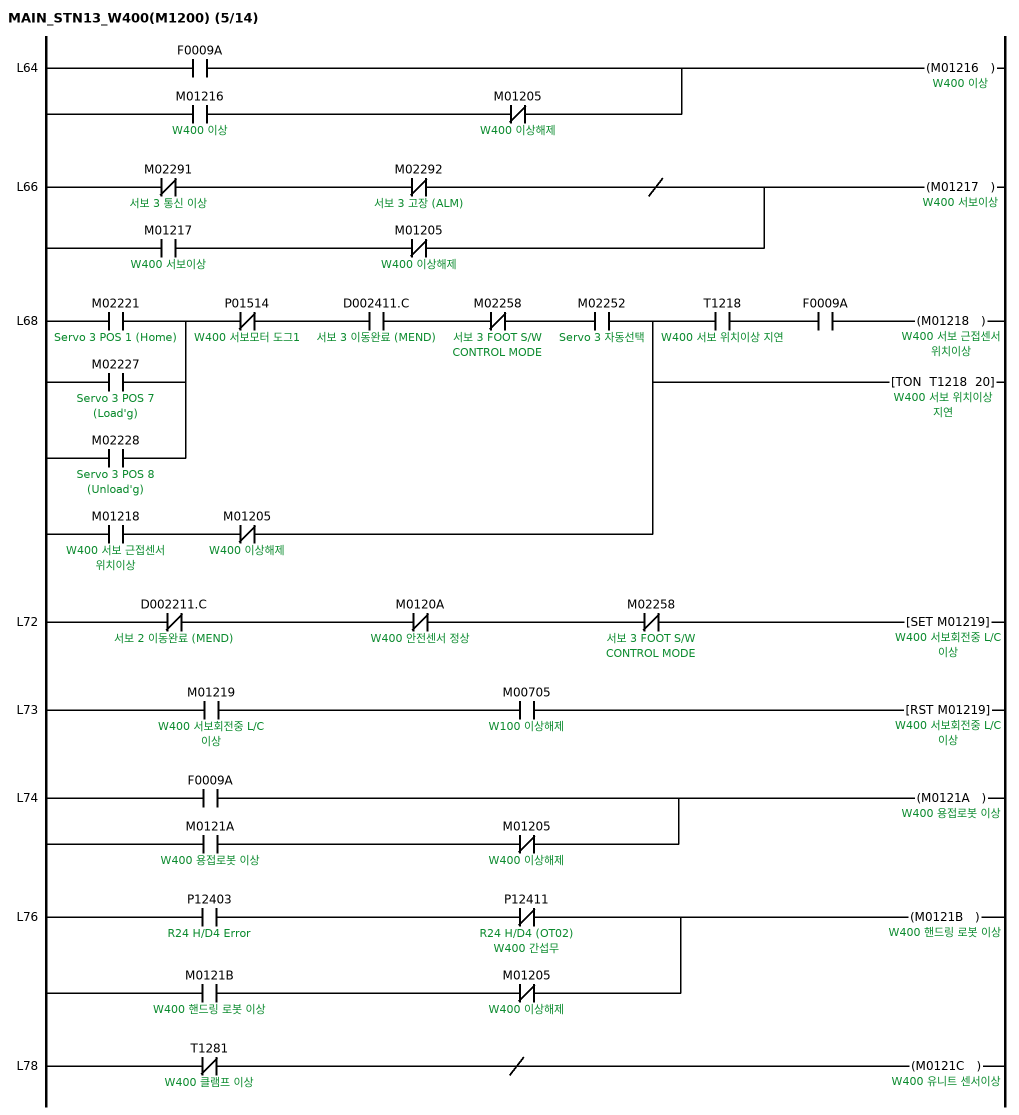
[picture p216: MAIN_STN13_W400(M1200) rungs L64-L78]
; L64
LOAD      F0009A
LOAD      M01216	// W400 이상
AND NOT   M01205	// W400 이상해제
OR LOAD
OUT       M01216	// W400 이상
; L66
LOAD NOT  M02291	// 서보 3 통신 이상
AND NOT   M02292	// 서보 3 고장 (ALM)
NOT
LOAD      M01217	// W400 서보이상
AND NOT   M01205	// W400 이상해제
OR LOAD
OUT       M01217	// W400 서보이상
; L68
LOAD      M02221	// Servo 3 POS 1 (Home)
OR        M02227	// Servo 3 POS 7 (Load'g)
OR        M02228	// Servo 3 POS 8 (Unload'g)
AND NOT   P01514	// W400 서보모터 도그1
AND       D002411.C	// 서보 3 이동완료 (MEND)
AND NOT   M02258	// 서보 3 FOOT S/W CONTROL MODE
AND       M02252	// Servo 3 자동선택
LOAD      M01218	// W400 서보 근접센서 위치이상
AND NOT   M01205	// W400 이상해제
OR LOAD
MPUSH
AND       T1218	// W400 서보 위치이상 지연
AND       F0009A
OUT       M01218	// W400 서보 근접센서 위치이상
MPOP
TON       T1218 20	// W400 서보 위치이상 지연
; L72
LOAD NOT  D002211.C	// 서보 2 이동완료 (MEND)
AND NOT   M0120A	// W400 안전센서 정상
AND NOT   M02258	// 서보 3 FOOT S/W CONTROL MODE
SET       M01219	// W400 서보회전중 L/C 이상
; L73
LOAD      M01219	// W400 서보회전중 L/C 이상
AND       M00705	// W100 이상해제
RST       M01219	// W400 서보회전중 L/C 이상
; L74
LOAD      F0009A
LOAD      M0121A	// W400 용접로봇 이상
AND NOT   M01205	// W400 이상해제
OR LOAD
OUT       M0121A	// W400 용접로봇 이상
; L76
LOAD      P12403	// R24 H/D4 Error
AND NOT   P12411	// R24 H/D4 (OT02) W400 간섭무
LOAD      M0121B	// W400 핸드링 로봇 이상
AND NOT   M01205	// W400 이상해제
OR LOAD
OUT       M0121B	// W400 핸드링 로봇 이상
; L78
LOAD NOT  T1281	// W400 클램프 이상
NOT
OUT       M0121C	// W400 유니트 센서이상

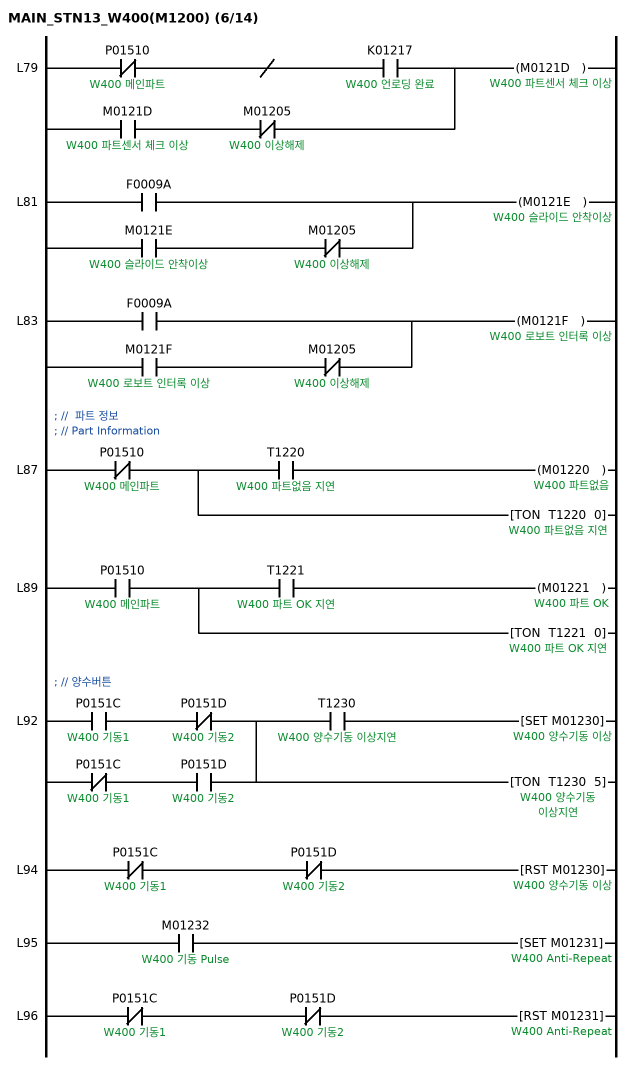
; L79
LOAD NOT  P01510	// W400 메인파트
NOT
AND       K01217	// W400 언로딩 완료
LOAD      M0121D	// W400 파트센서 체크 이상
AND NOT   M01205	// W400 이상해제
OR LOAD
OUT       M0121D	// W400 파트센서 체크 이상
; L81
LOAD      F0009A
LOAD      M0121E	// W400 슬라이드 안착이상
AND NOT   M01205	// W400 이상해제
OR LOAD
OUT       M0121E	// W400 슬라이드 안착이상
; L83
LOAD      F0009A
LOAD      M0121F	// W400 로보트 인터록 이상
AND NOT   M01205	// W400 이상해제
OR LOAD
OUT       M0121F	// W400 로보트 인터록 이상
//   //  파트 정보
//   // Part Information
; L87
LOAD NOT  P01510	// W400 메인파트
MPUSH
AND       T1220	// W400 파트없음 지연
OUT       M01220	// W400 파트없음
MPOP
TON       T1220 0	// W400 파트없음 지연
; L89
LOAD      P01510	// W400 메인파트
MPUSH
AND       T1221	// W400 파트 OK 지연
OUT       M01221	// W400 파트 OK
MPOP
TON       T1221 0	// W400 파트 OK 지연
//   // 양수버튼
; L92
LOAD      P0151C	// W400 기동1
AND NOT   P0151D	// W400 기동2
LOAD NOT  P0151C	// W400 기동1
AND       P0151D	// W400 기동2
OR LOAD
MPUSH
AND       T1230	// W400 양수기동 이상지연
SET       M01230	// W400 양수기동 이상
MPOP
TON       T1230 5	// W400 양수기동 이상지연
; L94
LOAD NOT  P0151C	// W400 기동1
AND NOT   P0151D	// W400 기동2
RST       M01230	// W400 양수기동 이상
; L95
LOAD      M01232	// W400 기동 Pulse
SET       M01231	// W400 Anti-Repeat
; L96
LOAD NOT  P0151C	// W400 기동1
AND NOT   P0151D	// W400 기동2
RST       M01231	// W400 Anti-Repeat

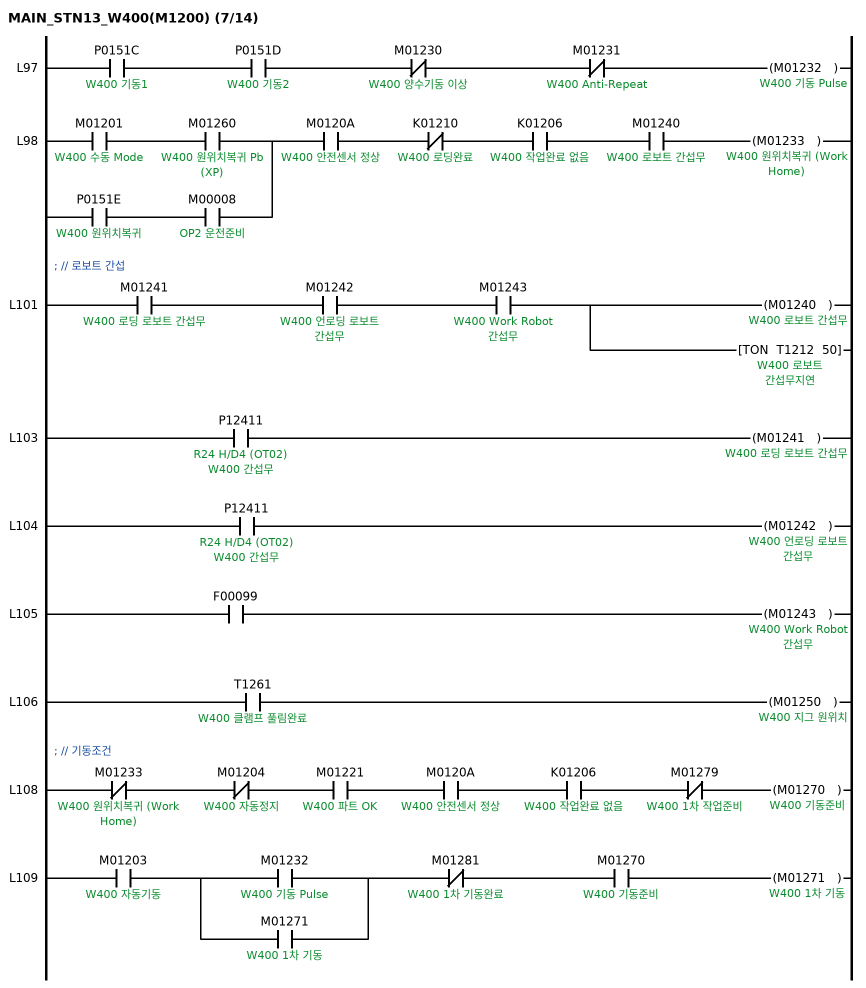
; L97
LOAD      P0151C	// W400 기동1
AND       P0151D	// W400 기동2
AND NOT   M01230	// W400 양수기동 이상
AND NOT   M01231	// W400 Anti-Repeat
OUT       M01232	// W400 기동 Pulse
; L98
LOAD      M01201	// W400 수동 Mode
AND       M01260	// W400 원위치복귀 Pb (XP)
LOAD      P0151E	// W400 원위치복귀
AND       M00008	// OP2 운전준비
OR LOAD
AND       M0120A	// W400 안전센서 정상
AND NOT   K01210	// W400 로딩완료
AND       K01206	// W400 작업완료 없음
AND       M01240	// W400 로보트 간섭무
OUT       M01233	// W400 원위치복귀 (Work Home)
//   // 로보트 간섭
; L101
LOAD      M01241	// W400 로딩 로보트 간섭무
AND       M01242	// W400 언로딩 로보트 간섭무
AND       M01243	// W400 Work Robot 간섭무
OUT       M01240	// W400 로보트 간섭무
TON       T1212 50	// W400 로보트 간섭무지연
; L103
LOAD      P12411	// R24 H/D4 (OT02) W400 간섭무
OUT       M01241	// W400 로딩 로보트 간섭무
; L104
LOAD      P12411	// R24 H/D4 (OT02) W400 간섭무
OUT       M01242	// W400 언로딩 로보트 간섭무
; L105
LOAD      F00099
OUT       M01243	// W400 Work Robot 간섭무
; L106
LOAD      T1261	// W400 클램프 풀림완료
OUT       M01250	// W400 지그 원위치
//   // 기동조건
; L108
LOAD NOT  M01233	// W400 원위치복귀 (Work Home)
AND NOT   M01204	// W400 자동정지
AND       M01221	// W400 파트 OK
AND       M0120A	// W400 안전센서 정상
AND       K01206	// W400 작업완료 없음
AND NOT   M01279	// W400 1차 작업준비
OUT       M01270	// W400 기동준비
; L109
LOAD      M01203	// W400 자동기동
LOAD      M01232	// W400 기동 Pulse
OR        M01271	// W400 1차 기동
AND LOAD
AND NOT   M01281	// W400 1차 기동완료
AND       M01270	// W400 기동준비
OUT       M01271	// W400 1차 기동

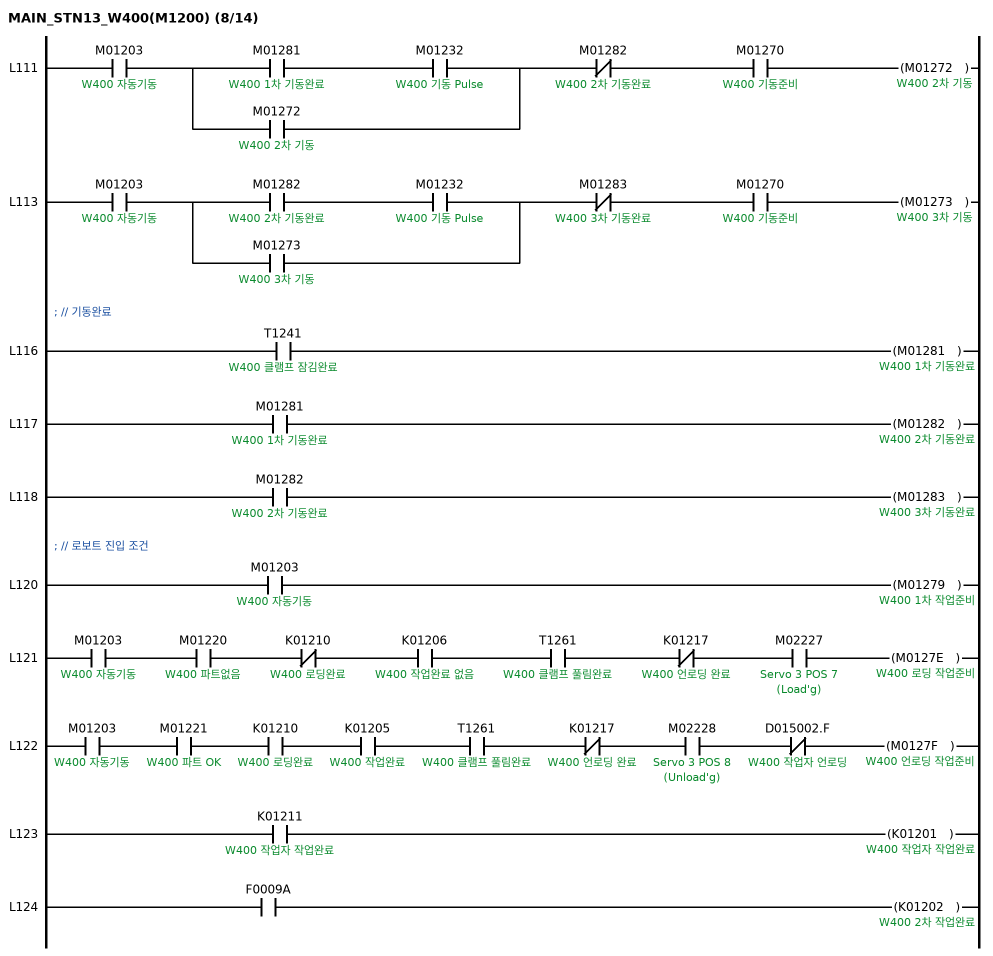
; L111
LOAD      M01203	// W400 자동기동
LOAD      M01281	// W400 1차 기동완료
AND       M01232	// W400 기동 Pulse
OR        M01272	// W400 2차 기동
AND LOAD
AND NOT   M01282	// W400 2차 기동완료
AND       M01270	// W400 기동준비
OUT       M01272	// W400 2차 기동
; L113
LOAD      M01203	// W400 자동기동
LOAD      M01282	// W400 2차 기동완료
AND       M01232	// W400 기동 Pulse
OR        M01273	// W400 3차 기동
AND LOAD
AND NOT   M01283	// W400 3차 기동완료
AND       M01270	// W400 기동준비
OUT       M01273	// W400 3차 기동
//   // 기동완료
; L116
LOAD      T1241	// W400 클램프 잠김완료
OUT       M01281	// W400 1차 기동완료
; L117
LOAD      M01281	// W400 1차 기동완료
OUT       M01282	// W400 2차 기동완료
; L118
LOAD      M01282	// W400 2차 기동완료
OUT       M01283	// W400 3차 기동완료
//   // 로보트 진입 조건
; L120
LOAD      M01203	// W400 자동기동
OUT       M01279	// W400 1차 작업준비
; L121
LOAD      M01203	// W400 자동기동
AND       M01220	// W400 파트없음
AND NOT   K01210	// W400 로딩완료
AND       K01206	// W400 작업완료 없음
AND       T1261	// W400 클램프 풀림완료
AND NOT   K01217	// W400 언로딩 완료
AND       M02227	// Servo 3 POS 7 (Load'g)
OUT       M0127E	// W400 로딩 작업준비
; L122
LOAD      M01203	// W400 자동기동
AND       M01221	// W400 파트 OK
AND       K01210	// W400 로딩완료
AND       K01205	// W400 작업완료
AND       T1261	// W400 클램프 풀림완료
AND NOT   K01217	// W400 언로딩 완료
AND       M02228	// Servo 3 POS 8 (Unload'g)
AND NOT   D015002.F	// W400 작업자 언로딩
OUT       M0127F	// W400 언로딩 작업준비
; L123
LOAD      K01211	// W400 작업자 작업완료
OUT       K01201	// W400 작업자 작업완료
; L124
LOAD      F0009A
OUT       K01202	// W400 2차 작업완료

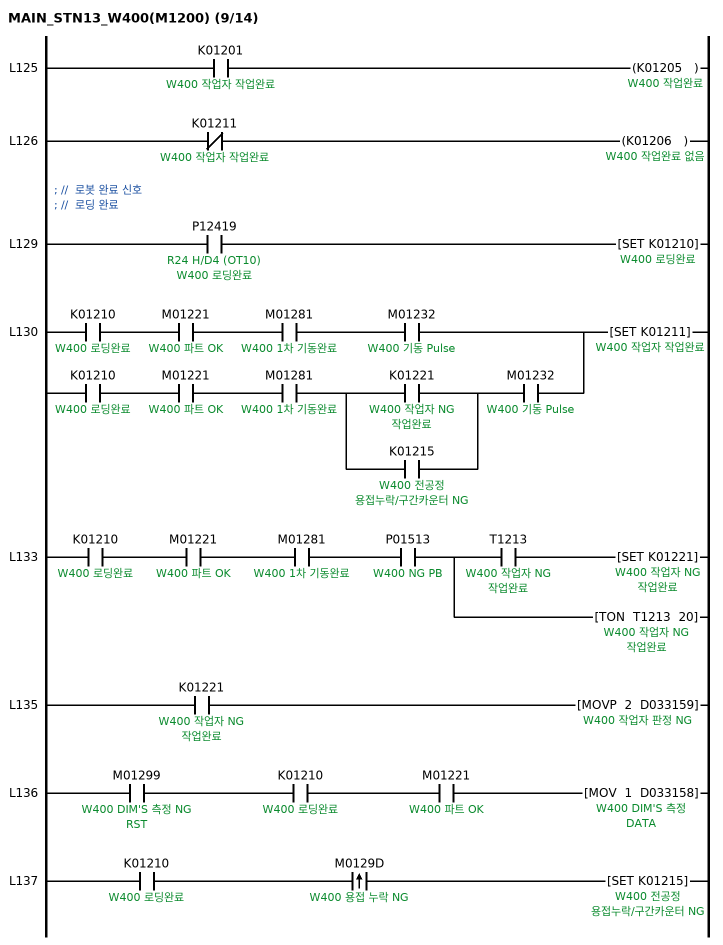
; L125
LOAD      K01201	// W400 작업자 작업완료
OUT       K01205	// W400 작업완료
; L126
LOAD NOT  K01211	// W400 작업자 작업완료
OUT       K01206	// W400 작업완료 없음
//   //  로봇 완료 신호
//   //  로딩 완료
; L129
LOAD      P12419	// R24 H/D4 (OT10) W400 로딩완료
SET       K01210	// W400 로딩완료
; L130
LOAD      K01210	// W400 로딩완료
AND       M01221	// W400 파트 OK
AND       M01281	// W400 1차 기동완료
AND       M01232	// W400 기동 Pulse
LOAD      K01210	// W400 로딩완료
AND       M01221	// W400 파트 OK
AND       M01281	// W400 1차 기동완료
LOAD      K01221	// W400 작업자 NG 작업완료
OR        K01215	// W400 전공정 용접누락/구간카운터 NG
AND LOAD
AND       M01232	// W400 기동 Pulse
OR LOAD
SET       K01211	// W400 작업자 작업완료
; L133
LOAD      K01210	// W400 로딩완료
AND       M01221	// W400 파트 OK
AND       M01281	// W400 1차 기동완료
AND       P01513	// W400 NG PB
MPUSH
AND       T1213	// W400 작업자 NG 작업완료
SET       K01221	// W400 작업자 NG 작업완료
MPOP
TON       T1213 20	// W400 작업자 NG 작업완료
; L135
LOAD      K01221	// W400 작업자 NG 작업완료
MOVP      2 D033159	// W400 작업자 판정 NG
; L136
LOAD      M01299	// W400 DIM'S 측정 NG RST
AND       K01210	// W400 로딩완료
AND       M01221	// W400 파트 OK
MOV       1 D033158	// W400 DIM'S 측정 DATA
; L137
LOAD      K01210	// W400 로딩완료
ANDP      M0129D	// W400 용접 누락 NG
SET       K01215	// W400 전공정 용접누락/구간카운터 NG

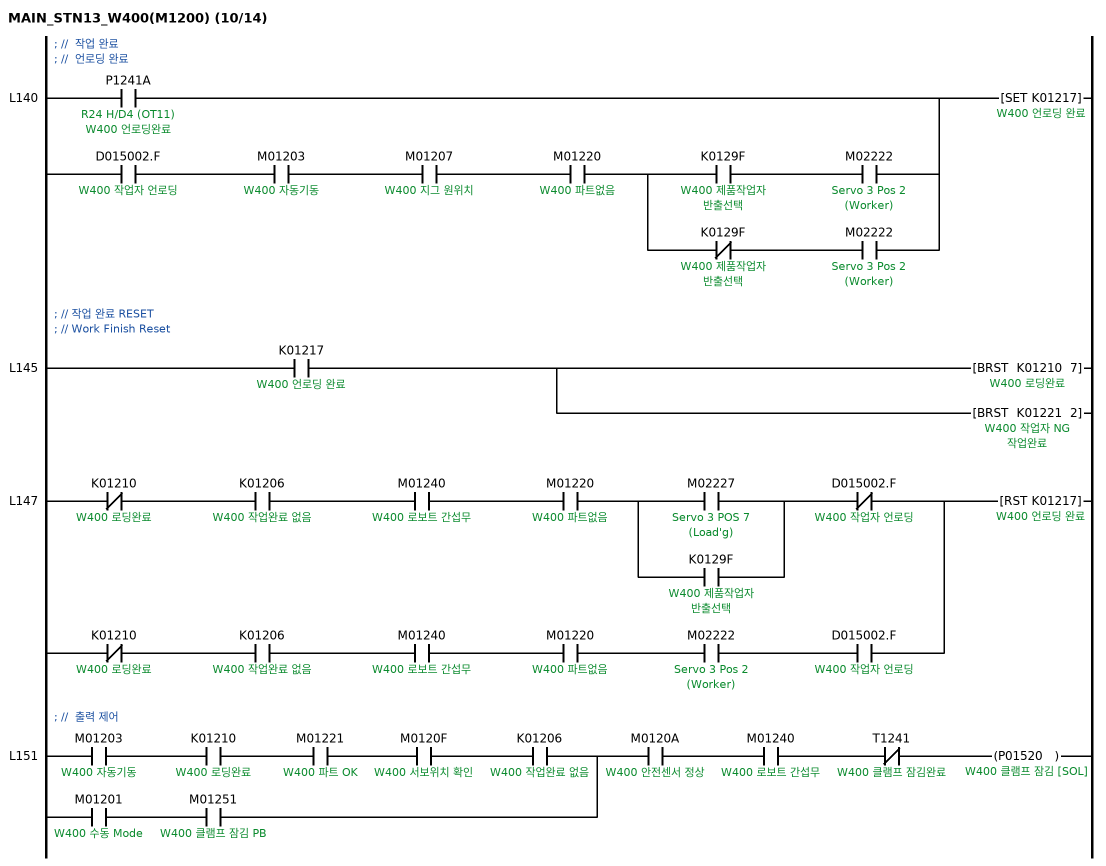
//   //  작업 완료
//   //  언로딩 완료
; L140
LOAD      P1241A	// R24 H/D4 (OT11) W400 언로딩완료
LOAD      D015002.F	// W400 작업자 언로딩
AND       M01203	// W400 자동기동
AND       M01207	// W400 지그 원위치
AND       M01220	// W400 파트없음
LOAD      K0129F	// W400 제품작업자 반출선택
AND       M02222	// Servo 3 Pos 2 (Worker)
LOAD NOT  K0129F	// W400 제품작업자 반출선택
AND       M02222	// Servo 3 Pos 2 (Worker)
OR LOAD
AND LOAD
OR LOAD
SET       K01217	// W400 언로딩 완료
//     // 작업 완료 RESET
//   // Work Finish Reset
; L145
LOAD      K01217	// W400 언로딩 완료
BRST      K01210 7	// W400 로딩완료
BRST      K01221 2	// W400 작업자 NG 작업완료
; L147
LOAD NOT  K01210	// W400 로딩완료
AND       K01206	// W400 작업완료 없음
AND       M01240	// W400 로보트 간섭무
AND       M01220	// W400 파트없음
LOAD      M02227	// Servo 3 POS 7 (Load'g)
OR        K0129F	// W400 제품작업자 반출선택
AND LOAD
AND NOT   D015002.F	// W400 작업자 언로딩
LOAD NOT  K01210	// W400 로딩완료
AND       K01206	// W400 작업완료 없음
AND       M01240	// W400 로보트 간섭무
AND       M01220	// W400 파트없음
AND       M02222	// Servo 3 Pos 2 (Worker)
AND       D015002.F	// W400 작업자 언로딩
OR LOAD
RST       K01217	// W400 언로딩 완료
//     //  출력 제어
; L151
LOAD      M01203	// W400 자동기동
AND       K01210	// W400 로딩완료
AND       M01221	// W400 파트 OK
AND       M0120F	// W400 서보위치 확인
AND       K01206	// W400 작업완료 없음
LOAD      M01201	// W400 수동 Mode
AND       M01251	// W400 클램프 잠김 PB
OR LOAD
AND       M0120A	// W400 안전센서 정상
AND       M01240	// W400 로보트 간섭무
AND NOT   T1241	// W400 클램프 잠김완료
OUT       P01520	// W400 클램프 잠김 [SOL]

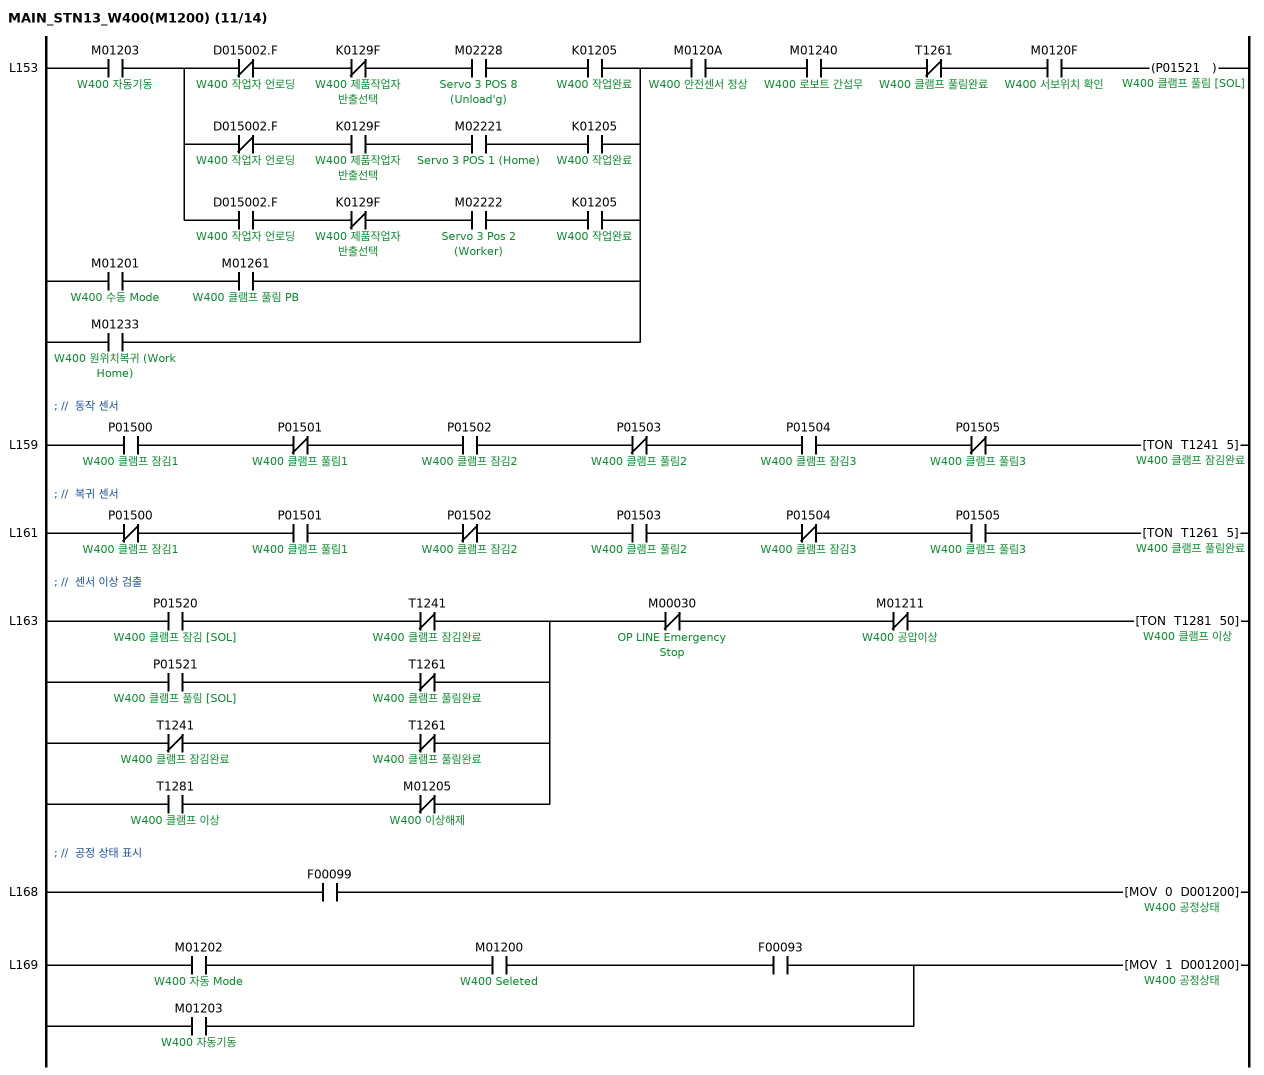
; L153
LOAD      M01203	// W400 자동기동
LOAD NOT  D015002.F	// W400 작업자 언로딩
AND NOT   K0129F	// W400 제품작업자 반출선택
AND       M02228	// Servo 3 POS 8 (Unload'g)
AND       K01205	// W400 작업완료
LOAD NOT  D015002.F	// W400 작업자 언로딩
AND       K0129F	// W400 제품작업자 반출선택
AND       M02221	// Servo 3 POS 1 (Home)
AND       K01205	// W400 작업완료
OR LOAD
LOAD      D015002.F	// W400 작업자 언로딩
AND NOT   K0129F	// W400 제품작업자 반출선택
AND       M02222	// Servo 3 Pos 2 (Worker)
AND       K01205	// W400 작업완료
OR LOAD
AND LOAD
LOAD      M01201	// W400 수동 Mode
AND       M01261	// W400 클램프 풀림 PB
OR LOAD
OR        M01233	// W400 원위치복귀 (Work Home)
AND       M0120A	// W400 안전센서 정상
AND       M01240	// W400 로보트 간섭무
AND NOT   T1261	// W400 클램프 풀림완료
AND       M0120F	// W400 서보위치 확인
OUT       P01521	// W400 클램프 풀림 [SOL]
//   //  동작 센서
; L159
LOAD      P01500	// W400 클램프 잠김1
AND NOT   P01501	// W400 클램프 풀림1
AND       P01502	// W400 클램프 잠김2
AND NOT   P01503	// W400 클램프 풀림2
AND       P01504	// W400 클램프 잠김3
AND NOT   P01505	// W400 클램프 풀림3
TON       T1241 5	// W400 클램프 잠김완료
//   //  복귀 센서
; L161
LOAD NOT  P01500	// W400 클램프 잠김1
AND       P01501	// W400 클램프 풀림1
AND NOT   P01502	// W400 클램프 잠김2
AND       P01503	// W400 클램프 풀림2
AND NOT   P01504	// W400 클램프 잠김3
AND       P01505	// W400 클램프 풀림3
TON       T1261 5	// W400 클램프 풀림완료
//     //  센서 이상 검출
; L163
LOAD      P01520	// W400 클램프 잠김 [SOL]
AND NOT   T1241	// W400 클램프 잠김완료
LOAD      P01521	// W400 클램프 풀림 [SOL]
AND NOT   T1261	// W400 클램프 풀림완료
OR LOAD
LOAD NOT  T1241	// W400 클램프 잠김완료
AND NOT   T1261	// W400 클램프 풀림완료
OR LOAD
LOAD      T1281	// W400 클램프 이상
AND NOT   M01205	// W400 이상해제
OR LOAD
AND NOT   M00030	// OP LINE Emergency Stop
AND NOT   M01211	// W400 공압이상
TON       T1281 50	// W400 클램프 이상
//   //  공정 상태 표시
; L168
LOAD      F00099
MOV       0 D001200	// W400 공정상태
; L169
LOAD      M01202	// W400 자동 Mode
AND       M01200	// W400 Seleted
AND       F00093
OR        M01203	// W400 자동기동
MOV       1 D001200	// W400 공정상태

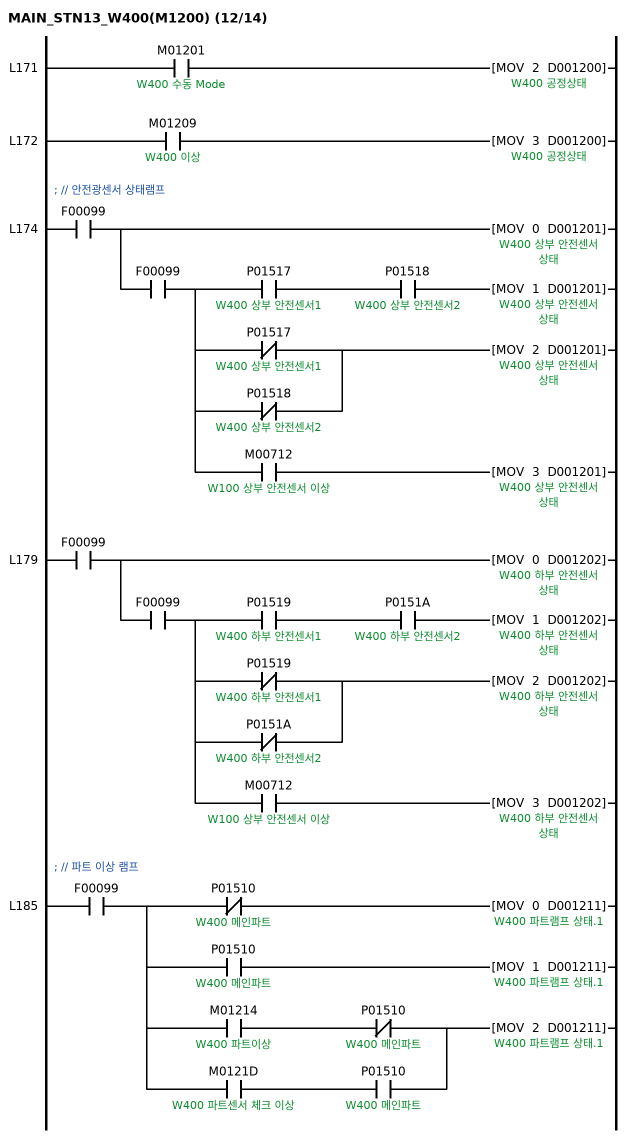
; L171
LOAD      M01201	// W400 수동 Mode
MOV       2 D001200	// W400 공정상태
; L172
LOAD      M01209	// W400 이상
MOV       3 D001200	// W400 공정상태
//   // 안전광센서 상태램프
; L174
LOAD      F00099
MOV       0 D001201	// W400 상부 안전센서 상태
AND       F00099
MPUSH
AND       P01517	// W400 상부 안전센서1
AND       P01518	// W400 상부 안전센서2
MOV       1 D001201	// W400 상부 안전센서 상태
MLOAD
LOAD NOT  P01517	// W400 상부 안전센서1
OR NOT    P01518	// W400 상부 안전센서2
AND LOAD
MOV       2 D001201	// W400 상부 안전센서 상태
MPOP
AND       M00712	// W100 상부 안전센서 이상
MOV       3 D001201	// W400 상부 안전센서 상태
; L179
LOAD      F00099
MOV       0 D001202	// W400 하부 안전센서 상태
AND       F00099
MPUSH
AND       P01519	// W400 하부 안전센서1
AND       P0151A	// W400 하부 안전센서2
MOV       1 D001202	// W400 하부 안전센서 상태
MLOAD
LOAD NOT  P01519	// W400 하부 안전센서1
OR NOT    P0151A	// W400 하부 안전센서2
AND LOAD
MOV       2 D001202	// W400 하부 안전센서 상태
MPOP
AND       M00712	// W100 상부 안전센서 이상
MOV       3 D001202	// W400 하부 안전센서 상태
//   // 파트 이상 램프
; L185
LOAD      F00099
MPUSH
AND NOT   P01510	// W400 메인파트
MOV       0 D001211	// W400 파트램프 상태.1
MLOAD
AND       P01510	// W400 메인파트
MOV       1 D001211	// W400 파트램프 상태.1
MPOP
LOAD      M01214	// W400 파트이상
AND NOT   P01510	// W400 메인파트
LOAD      M0121D	// W400 파트센서 체크 이상
AND       P01510	// W400 메인파트
OR LOAD
AND LOAD
MOV       2 D001211	// W400 파트램프 상태.1

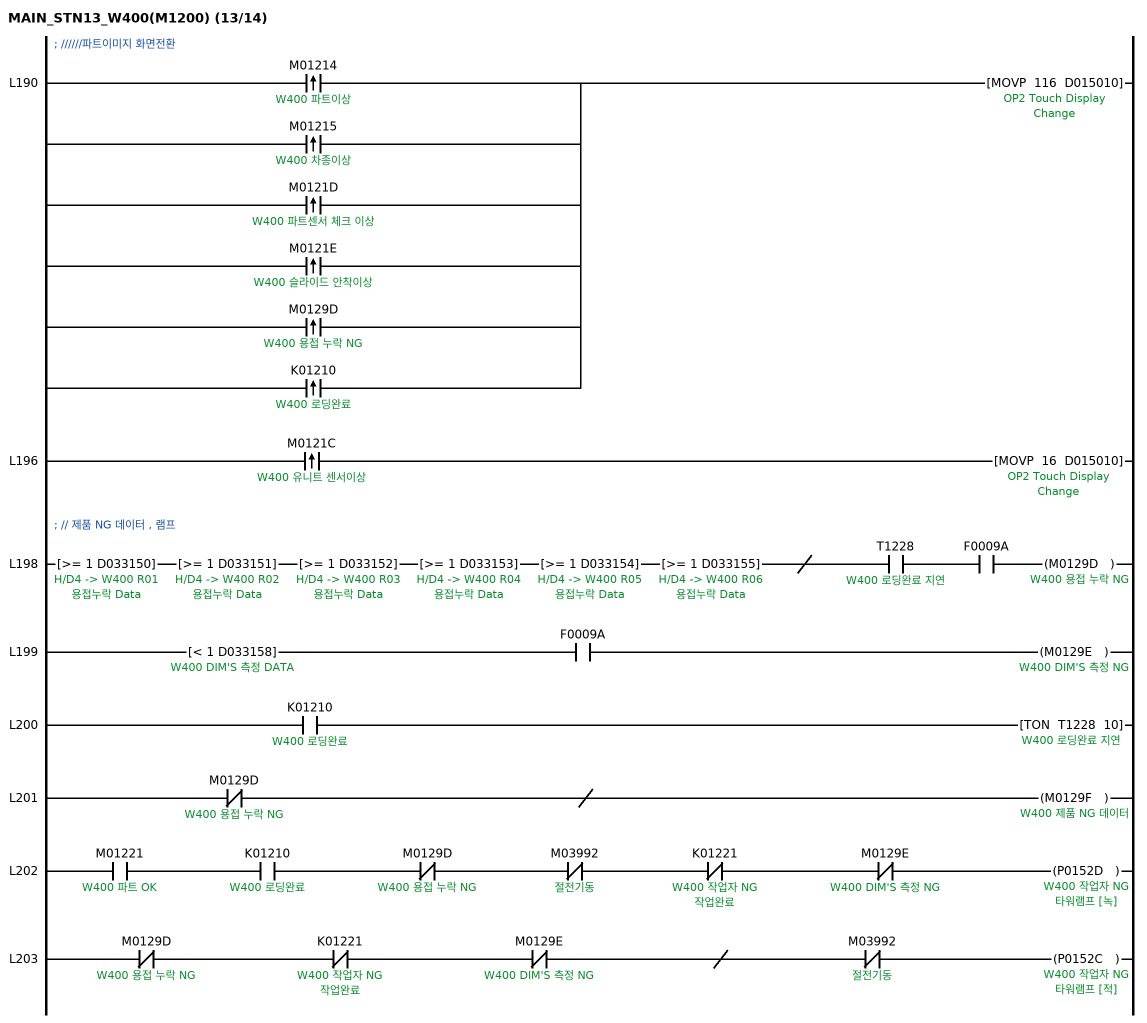
// //////파트이미지 화면전환
; L190
LOADP     M01214	// W400 파트이상
ORP       M01215	// W400 차종이상
ORP       M0121D	// W400 파트센서 체크 이상
ORP       M0121E	// W400 슬라이드 안착이상
ORP       M0129D	// W400 용접 누락 NG
ORP       K01210	// W400 로딩완료
MOVP      116 D015010	// OP2 Touch Display Change
; L196
LOADP     M0121C	// W400 유니트 센서이상
MOVP      16 D015010	// OP2 Touch Display Change
//   // 제품 NG 데이터 , 램프
; L198
LOAD>=    1 D033150	// H/D4 -> W400 R01 용접누락 Data
AND>=     1 D033151	// H/D4 -> W400 R02 용접누락 Data
AND>=     1 D033152	// H/D4 -> W400 R03 용접누락 Data
AND>=     1 D033153	// H/D4 -> W400 R04 용접누락 Data
AND>=     1 D033154	// H/D4 -> W400 R05 용접누락 Data
AND>=     1 D033155	// H/D4 -> W400 R06 용접누락 Data
NOT
AND       T1228	// W400 로딩완료 지연
AND       F0009A
OUT       M0129D	// W400 용접 누락 NG
; L199
LOAD<     1 D033158	// W400 DIM'S 측정 DATA
AND       F0009A
OUT       M0129E	// W400 DIM'S 측정 NG
; L200
LOAD      K01210	// W400 로딩완료
TON       T1228 10	// W400 로딩완료 지연
; L201
LOAD NOT  M0129D	// W400 용접 누락 NG
NOT
OUT       M0129F	// W400 제품 NG 데이터
; L202
LOAD      M01221	// W400 파트 OK
AND       K01210	// W400 로딩완료
AND NOT   M0129D	// W400 용접 누락 NG
AND NOT   M03992	// 절전기동
AND NOT   K01221	// W400 작업자 NG 작업완료
AND NOT   M0129E	// W400 DIM'S 측정 NG
OUT       P0152D	// W400 작업자 NG 타워램프 [녹]
; L203
LOAD NOT  M0129D	// W400 용접 누락 NG
AND NOT   K01221	// W400 작업자 NG 작업완료
AND NOT   M0129E	// W400 DIM'S 측정 NG
NOT
AND NOT   M03992	// 절전기동
OUT       P0152C	// W400 작업자 NG 타워램프 [적]

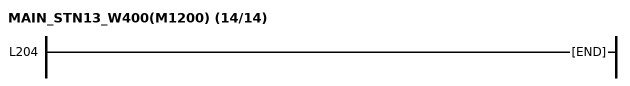
; L204
END

PROGRAM MAIN_STN14_W450(M1300) (task: 스캔 프로그램)

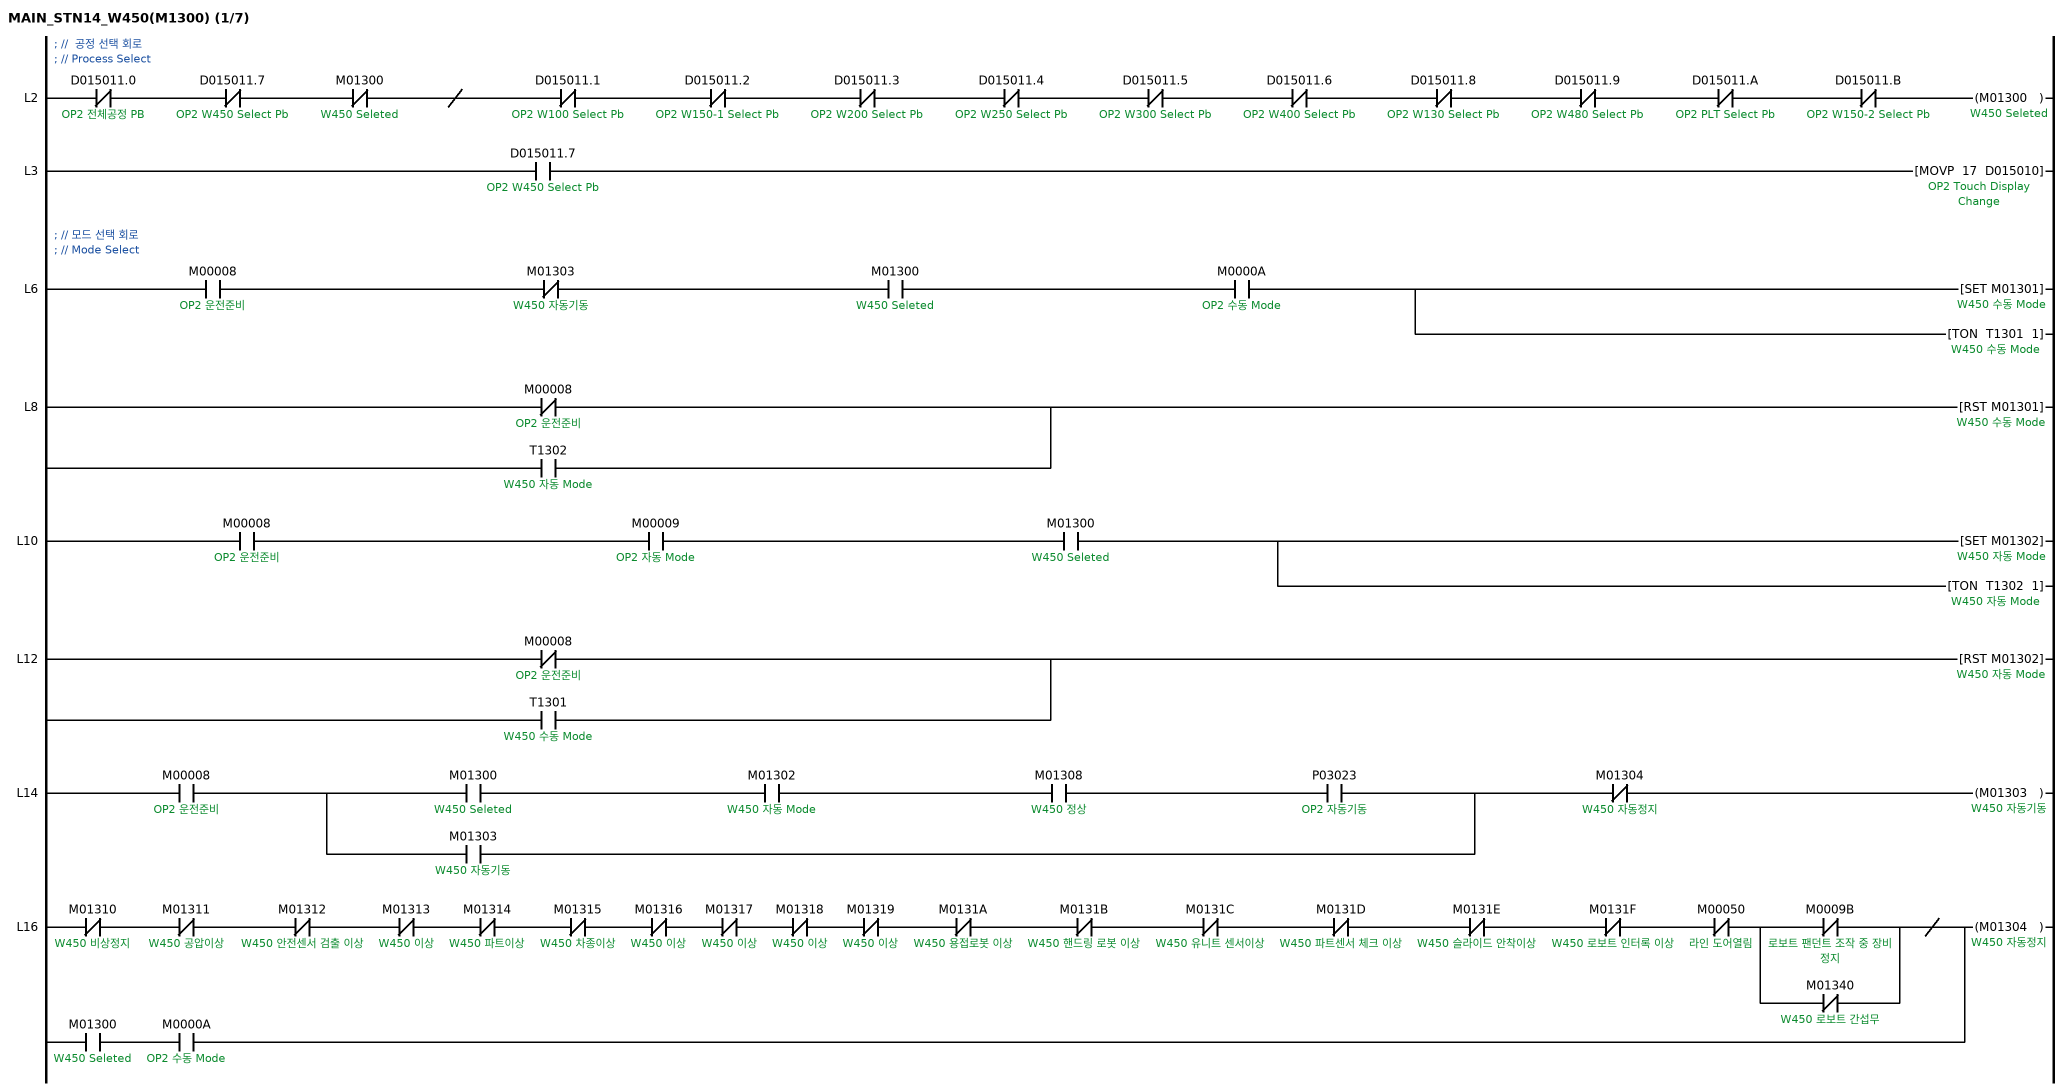
//   //  공정 선택 회로
//   // Process Select
; L2
LOAD NOT  D015011.0	// OP2 전체공정 PB
AND NOT   D015011.7	// OP2 W450 Select Pb
AND NOT   M01300	// W450 Seleted
NOT
AND NOT   D015011.1	// OP2 W100 Select Pb
AND NOT   D015011.2	// OP2 W150-1 Select Pb
AND NOT   D015011.3	// OP2 W200 Select Pb
AND NOT   D015011.4	// OP2 W250 Select Pb
AND NOT   D015011.5	// OP2 W300 Select Pb
AND NOT   D015011.6	// OP2 W400 Select Pb
AND NOT   D015011.8	// OP2 W130 Select Pb
AND NOT   D015011.9	// OP2 W480 Select Pb
AND NOT   D015011.A	// OP2 PLT Select Pb
AND NOT   D015011.B	// OP2 W150-2 Select Pb
OUT       M01300	// W450 Seleted
; L3
LOAD      D015011.7	// OP2 W450 Select Pb
MOVP      17 D015010	// OP2 Touch Display Change
// // 모드 선택 회로
//   // Mode Select
; L6
LOAD      M00008	// OP2 운전준비
AND NOT   M01303	// W450 자동기동
AND       M01300	// W450 Seleted
AND       M0000A	// OP2 수동 Mode
SET       M01301	// W450 수동 Mode
TON       T1301 1	// W450 수동 Mode
; L8
LOAD NOT  M00008	// OP2 운전준비
OR        T1302	// W450 자동 Mode
RST       M01301	// W450 수동 Mode
; L10
LOAD      M00008	// OP2 운전준비
AND       M00009	// OP2 자동 Mode
AND       M01300	// W450 Seleted
SET       M01302	// W450 자동 Mode
TON       T1302 1	// W450 자동 Mode
; L12
LOAD NOT  M00008	// OP2 운전준비
OR        T1301	// W450 수동 Mode
RST       M01302	// W450 자동 Mode
; L14
LOAD      M00008	// OP2 운전준비
LOAD      M01300	// W450 Seleted
AND       M01302	// W450 자동 Mode
AND       M01308	// W450 정상
AND       P03023	// OP2 자동기동
OR        M01303	// W450 자동기동
AND LOAD
AND NOT   M01304	// W450 자동정지
OUT       M01303	// W450 자동기동
; L16
LOAD NOT  M01310	// W450 비상정지
AND NOT   M01311	// W450 공압이상
AND NOT   M01312	// W450 안전센서 검출 이상
AND NOT   M01313	// W450 이상
AND NOT   M01314	// W450 파트이상
AND NOT   M01315	// W450 차종이상
AND NOT   M01316	// W450 이상
AND NOT   M01317	// W450 이상
AND NOT   M01318	// W450 이상
AND NOT   M01319	// W450 이상
AND NOT   M0131A	// W450 용접로봇 이상
AND NOT   M0131B	// W450 핸드링 로봇 이상
AND NOT   M0131C	// W450 유니트 센서이상
AND NOT   M0131D	// W450 파트센서 체크 이상
AND NOT   M0131E	// W450 슬라이드 안착이상
AND NOT   M0131F	// W450 로보트 인터록 이상
AND NOT   M00050	// 라인 도어열림
LOAD NOT  M0009B	// 로보트 팬던트 조작 중 장비 정지
OR NOT    M01340	// W450 로보트 간섭무
AND LOAD
NOT
LOAD      M01300	// W450 Seleted
AND       M0000A	// OP2 수동 Mode
OR LOAD
OUT       M01304	// W450 자동정지

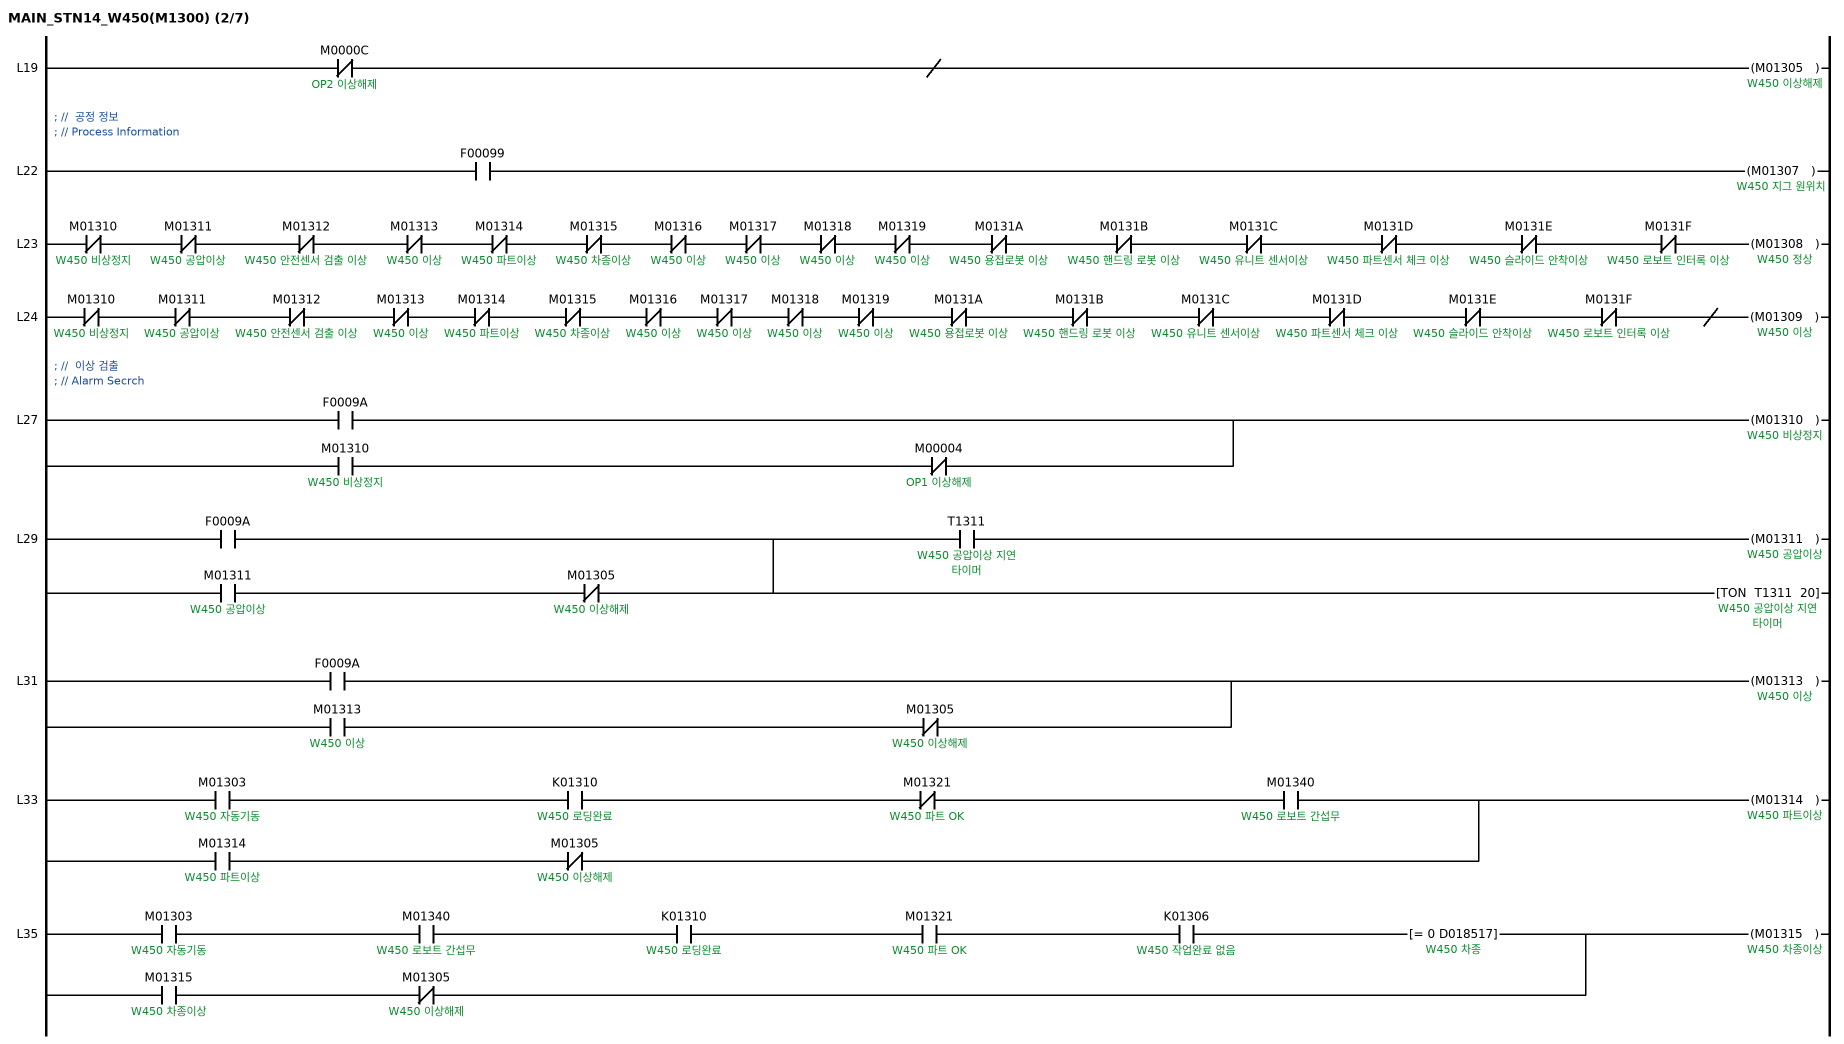
; L19
LOAD NOT  M0000C	// OP2 이상해제
NOT
OUT       M01305	// W450 이상해제
//   //  공정 정보
//   // Process Information
; L22
LOAD      F00099
OUT       M01307	// W450 지그 원위치
; L23
LOAD NOT  M01310	// W450 비상정지
AND NOT   M01311	// W450 공압이상
AND NOT   M01312	// W450 안전센서 검출 이상
AND NOT   M01313	// W450 이상
AND NOT   M01314	// W450 파트이상
AND NOT   M01315	// W450 차종이상
AND NOT   M01316	// W450 이상
AND NOT   M01317	// W450 이상
AND NOT   M01318	// W450 이상
AND NOT   M01319	// W450 이상
AND NOT   M0131A	// W450 용접로봇 이상
AND NOT   M0131B	// W450 핸드링 로봇 이상
AND NOT   M0131C	// W450 유니트 센서이상
AND NOT   M0131D	// W450 파트센서 체크 이상
AND NOT   M0131E	// W450 슬라이드 안착이상
AND NOT   M0131F	// W450 로보트 인터록 이상
OUT       M01308	// W450 정상
; L24
LOAD NOT  M01310	// W450 비상정지
AND NOT   M01311	// W450 공압이상
AND NOT   M01312	// W450 안전센서 검출 이상
AND NOT   M01313	// W450 이상
AND NOT   M01314	// W450 파트이상
AND NOT   M01315	// W450 차종이상
AND NOT   M01316	// W450 이상
AND NOT   M01317	// W450 이상
AND NOT   M01318	// W450 이상
AND NOT   M01319	// W450 이상
AND NOT   M0131A	// W450 용접로봇 이상
AND NOT   M0131B	// W450 핸드링 로봇 이상
AND NOT   M0131C	// W450 유니트 센서이상
AND NOT   M0131D	// W450 파트센서 체크 이상
AND NOT   M0131E	// W450 슬라이드 안착이상
AND NOT   M0131F	// W450 로보트 인터록 이상
NOT
OUT       M01309	// W450 이상
//   //  이상 검출
//   // Alarm Secrch
; L27
LOAD      F0009A
LOAD      M01310	// W450 비상정지
AND NOT   M00004	// OP1 이상해제
OR LOAD
OUT       M01310	// W450 비상정지
; L29
LOAD      F0009A
LOAD      M01311	// W450 공압이상
AND NOT   M01305	// W450 이상해제
OR LOAD
MPUSH
AND       T1311	// W450 공압이상 지연 타이머
OUT       M01311	// W450 공압이상
MPOP
TON       T1311 20	// W450 공압이상 지연 타이머
; L31
LOAD      F0009A
LOAD      M01313	// W450 이상
AND NOT   M01305	// W450 이상해제
OR LOAD
OUT       M01313	// W450 이상
; L33
LOAD      M01303	// W450 자동기동
AND       K01310	// W450 로딩완료
AND NOT   M01321	// W450 파트 OK
AND       M01340	// W450 로보트 간섭무
LOAD      M01314	// W450 파트이상
AND NOT   M01305	// W450 이상해제
OR LOAD
OUT       M01314	// W450 파트이상
; L35
LOAD      M01303	// W450 자동기동
AND       M01340	// W450 로보트 간섭무
AND       K01310	// W450 로딩완료
AND       M01321	// W450 파트 OK
AND       K01306	// W450 작업완료 없음
AND=      0 D018517	// W450 차종
LOAD      M01315	// W450 차종이상
AND NOT   M01305	// W450 이상해제
OR LOAD
OUT       M01315	// W450 차종이상

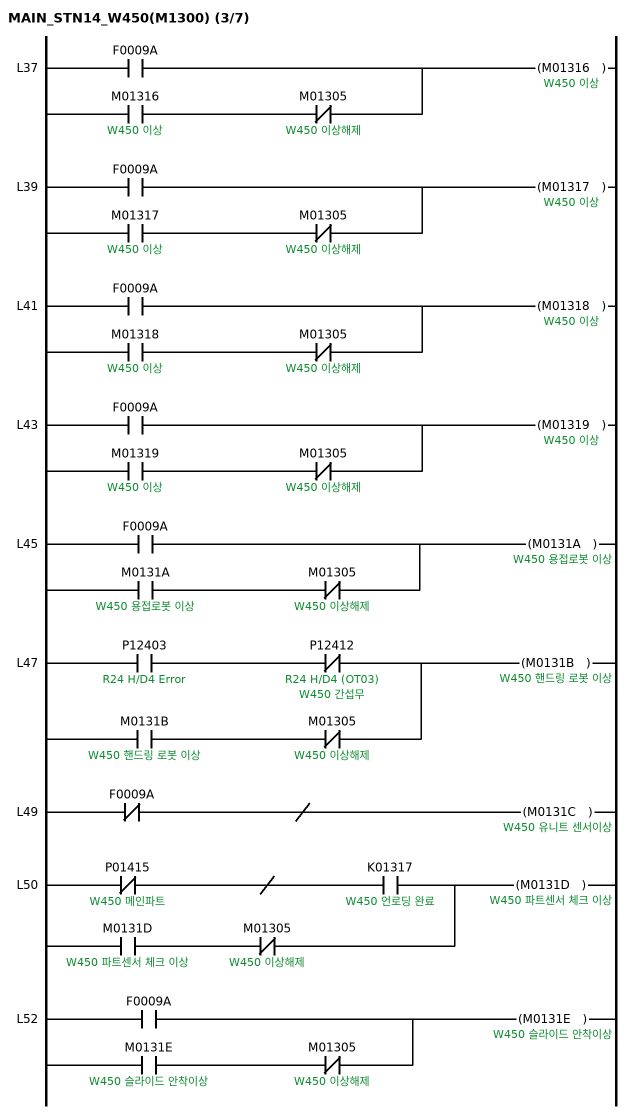
; L37
LOAD      F0009A
LOAD      M01316	// W450 이상
AND NOT   M01305	// W450 이상해제
OR LOAD
OUT       M01316	// W450 이상
; L39
LOAD      F0009A
LOAD      M01317	// W450 이상
AND NOT   M01305	// W450 이상해제
OR LOAD
OUT       M01317	// W450 이상
; L41
LOAD      F0009A
LOAD      M01318	// W450 이상
AND NOT   M01305	// W450 이상해제
OR LOAD
OUT       M01318	// W450 이상
; L43
LOAD      F0009A
LOAD      M01319	// W450 이상
AND NOT   M01305	// W450 이상해제
OR LOAD
OUT       M01319	// W450 이상
; L45
LOAD      F0009A
LOAD      M0131A	// W450 용접로봇 이상
AND NOT   M01305	// W450 이상해제
OR LOAD
OUT       M0131A	// W450 용접로봇 이상
; L47
LOAD      P12403	// R24 H/D4 Error
AND NOT   P12412	// R24 H/D4 (OT03) W450 간섭무
LOAD      M0131B	// W450 핸드링 로봇 이상
AND NOT   M01305	// W450 이상해제
OR LOAD
OUT       M0131B	// W450 핸드링 로봇 이상
; L49
LOAD NOT  F0009A
NOT
OUT       M0131C	// W450 유니트 센서이상
; L50
LOAD NOT  P01415	// W450 메인파트
NOT
AND       K01317	// W450 언로딩 완료
LOAD      M0131D	// W450 파트센서 체크 이상
AND NOT   M01305	// W450 이상해제
OR LOAD
OUT       M0131D	// W450 파트센서 체크 이상
; L52
LOAD      F0009A
LOAD      M0131E	// W450 슬라이드 안착이상
AND NOT   M01305	// W450 이상해제
OR LOAD
OUT       M0131E	// W450 슬라이드 안착이상

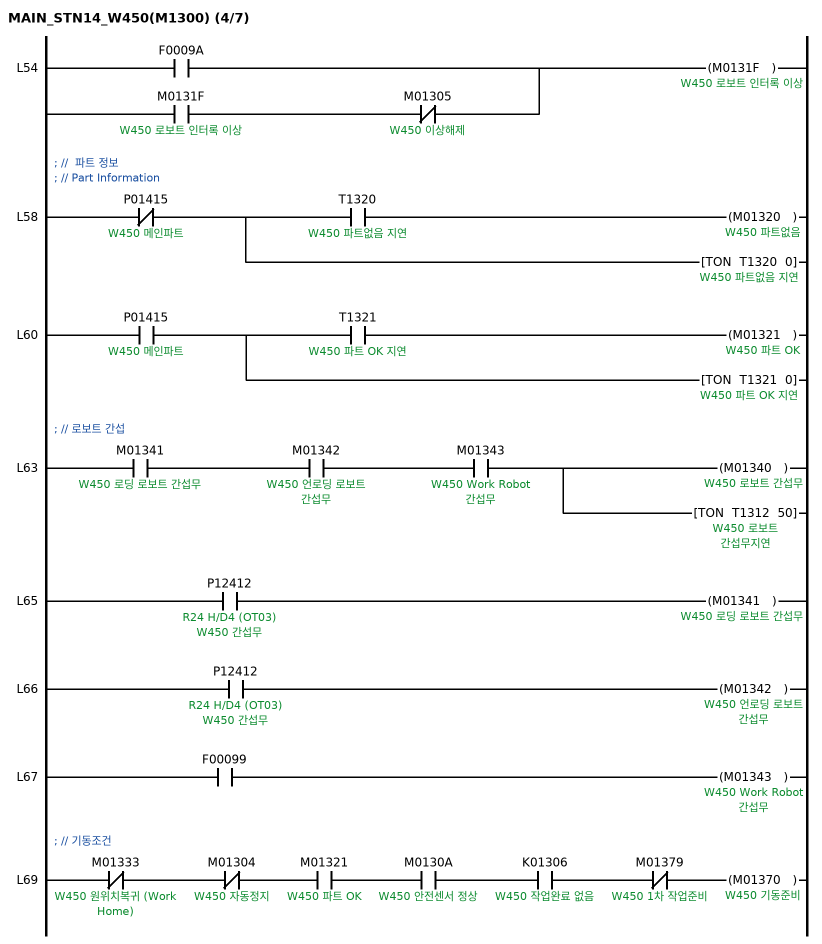
; L54
LOAD      F0009A
LOAD      M0131F	// W450 로보트 인터록 이상
AND NOT   M01305	// W450 이상해제
OR LOAD
OUT       M0131F	// W450 로보트 인터록 이상
//   //  파트 정보
//   // Part Information
; L58
LOAD NOT  P01415	// W450 메인파트
MPUSH
AND       T1320	// W450 파트없음 지연
OUT       M01320	// W450 파트없음
MPOP
TON       T1320 0	// W450 파트없음 지연
; L60
LOAD      P01415	// W450 메인파트
MPUSH
AND       T1321	// W450 파트 OK 지연
OUT       M01321	// W450 파트 OK
MPOP
TON       T1321 0	// W450 파트 OK 지연
//   // 로보트 간섭
; L63
LOAD      M01341	// W450 로딩 로보트 간섭무
AND       M01342	// W450 언로딩 로보트 간섭무
AND       M01343	// W450 Work Robot 간섭무
OUT       M01340	// W450 로보트 간섭무
TON       T1312 50	// W450 로보트 간섭무지연
; L65
LOAD      P12412	// R24 H/D4 (OT03) W450 간섭무
OUT       M01341	// W450 로딩 로보트 간섭무
; L66
LOAD      P12412	// R24 H/D4 (OT03) W450 간섭무
OUT       M01342	// W450 언로딩 로보트 간섭무
; L67
LOAD      F00099
OUT       M01343	// W450 Work Robot 간섭무
//   // 기동조건
; L69
LOAD NOT  M01333	// W450 원위치복귀 (Work Home)
AND NOT   M01304	// W450 자동정지
AND       M01321	// W450 파트 OK
AND       M0130A	// W450 안전센서 정상
AND       K01306	// W450 작업완료 없음
AND NOT   M01379	// W450 1차 작업준비
OUT       M01370	// W450 기동준비

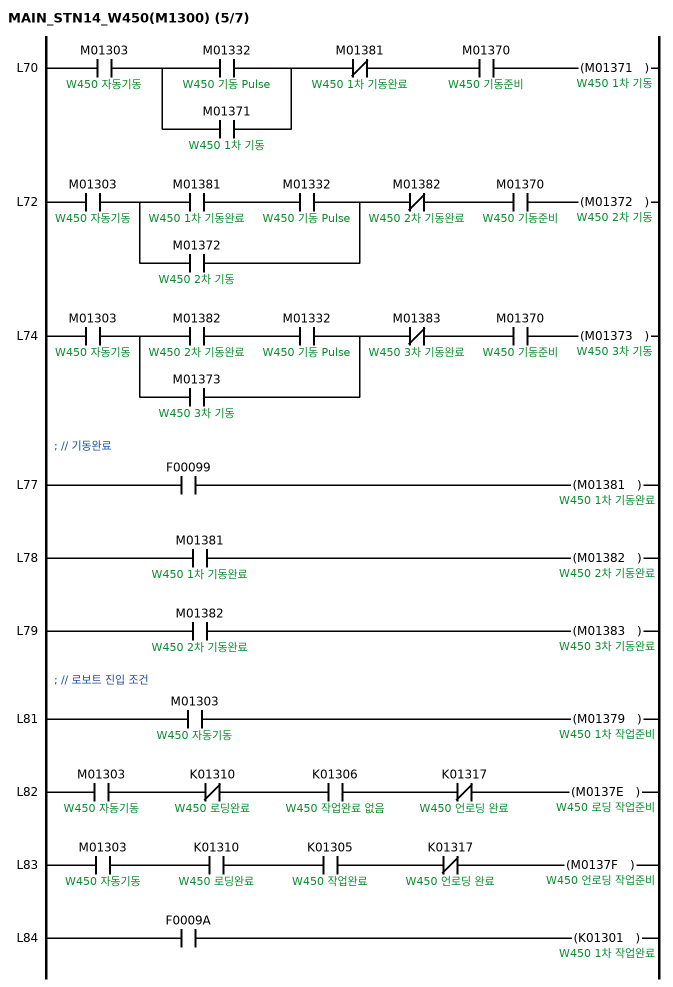
; L70
LOAD      M01303	// W450 자동기동
LOAD      M01332	// W450 기동 Pulse
OR        M01371	// W450 1차 기동
AND LOAD
AND NOT   M01381	// W450 1차 기동완료
AND       M01370	// W450 기동준비
OUT       M01371	// W450 1차 기동
; L72
LOAD      M01303	// W450 자동기동
LOAD      M01381	// W450 1차 기동완료
AND       M01332	// W450 기동 Pulse
OR        M01372	// W450 2차 기동
AND LOAD
AND NOT   M01382	// W450 2차 기동완료
AND       M01370	// W450 기동준비
OUT       M01372	// W450 2차 기동
; L74
LOAD      M01303	// W450 자동기동
LOAD      M01382	// W450 2차 기동완료
AND       M01332	// W450 기동 Pulse
OR        M01373	// W450 3차 기동
AND LOAD
AND NOT   M01383	// W450 3차 기동완료
AND       M01370	// W450 기동준비
OUT       M01373	// W450 3차 기동
//   // 기동완료
; L77
LOAD      F00099
OUT       M01381	// W450 1차 기동완료
; L78
LOAD      M01381	// W450 1차 기동완료
OUT       M01382	// W450 2차 기동완료
; L79
LOAD      M01382	// W450 2차 기동완료
OUT       M01383	// W450 3차 기동완료
//   // 로보트 진입 조건
; L81
LOAD      M01303	// W450 자동기동
OUT       M01379	// W450 1차 작업준비
; L82
LOAD      M01303	// W450 자동기동
AND NOT   K01310	// W450 로딩완료
AND       K01306	// W450 작업완료 없음
AND NOT   K01317	// W450 언로딩 완료
OUT       M0137E	// W450 로딩 작업준비
; L83
LOAD      M01303	// W450 자동기동
AND       K01310	// W450 로딩완료
AND       K01305	// W450 작업완료
AND NOT   K01317	// W450 언로딩 완료
OUT       M0137F	// W450 언로딩 작업준비
; L84
LOAD      F0009A
OUT       K01301	// W450 1차 작업완료

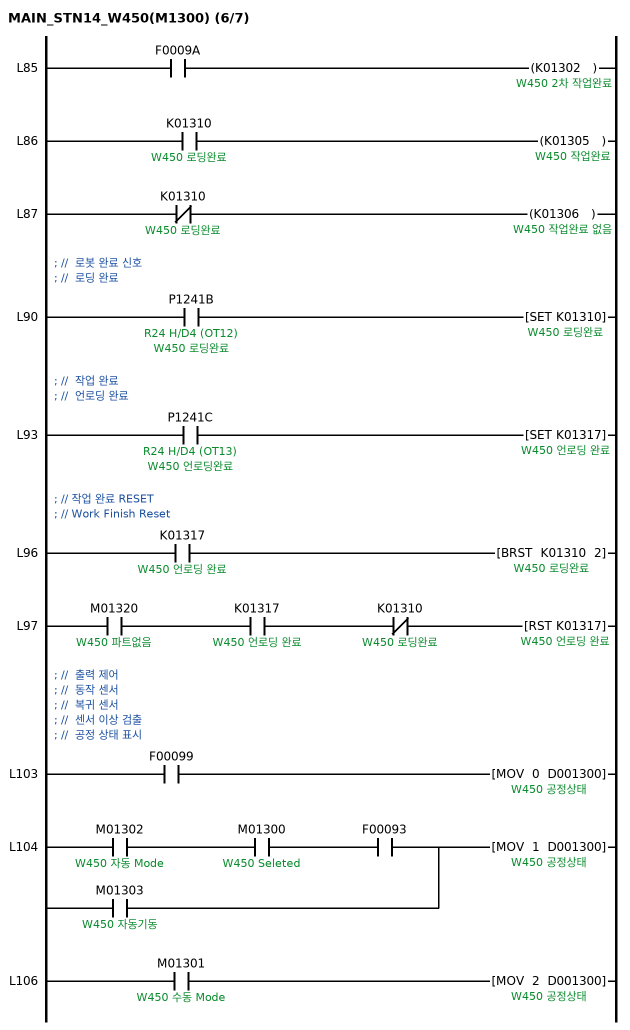
; L85
LOAD      F0009A
OUT       K01302	// W450 2차 작업완료
; L86
LOAD      K01310	// W450 로딩완료
OUT       K01305	// W450 작업완료
; L87
LOAD NOT  K01310	// W450 로딩완료
OUT       K01306	// W450 작업완료 없음
//   //  로봇 완료 신호
//   //  로딩 완료
; L90
LOAD      P1241B	// R24 H/D4 (OT12) W450 로딩완료
SET       K01310	// W450 로딩완료
//   //  작업 완료
//   //  언로딩 완료
; L93
LOAD      P1241C	// R24 H/D4 (OT13) W450 언로딩완료
SET       K01317	// W450 언로딩 완료
//     // 작업 완료 RESET
//   // Work Finish Reset
; L96
LOAD      K01317	// W450 언로딩 완료
BRST      K01310 2	// W450 로딩완료
; L97
LOAD      M01320	// W450 파트없음
AND       K01317	// W450 언로딩 완료
AND NOT   K01310	// W450 로딩완료
RST       K01317	// W450 언로딩 완료
//     //  출력 제어
//   //  동작 센서
//   //  복귀 센서
//     //  센서 이상 검출
//   //  공정 상태 표시
; L103
LOAD      F00099
MOV       0 D001300	// W450 공정상태
; L104
LOAD      M01302	// W450 자동 Mode
AND       M01300	// W450 Seleted
AND       F00093
OR        M01303	// W450 자동기동
MOV       1 D001300	// W450 공정상태
; L106
LOAD      M01301	// W450 수동 Mode
MOV       2 D001300	// W450 공정상태

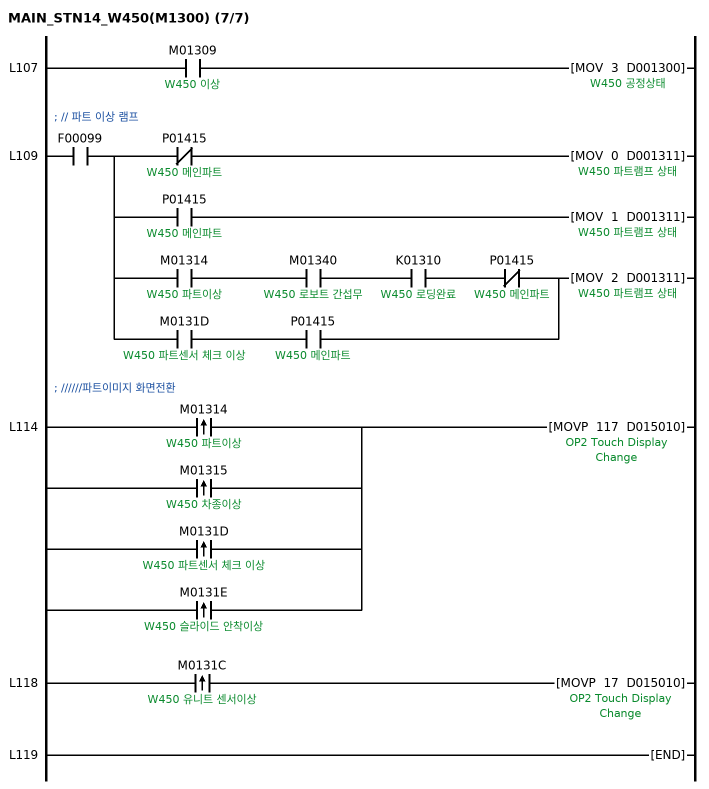
; L107
LOAD      M01309	// W450 이상
MOV       3 D001300	// W450 공정상태
//   // 파트 이상 램프
; L109
LOAD      F00099
MPUSH
AND NOT   P01415	// W450 메인파트
MOV       0 D001311	// W450 파트램프 상태
MLOAD
AND       P01415	// W450 메인파트
MOV       1 D001311	// W450 파트램프 상태
MPOP
LOAD      M01314	// W450 파트이상
AND       M01340	// W450 로보트 간섭무
AND       K01310	// W450 로딩완료
AND NOT   P01415	// W450 메인파트
LOAD      M0131D	// W450 파트센서 체크 이상
AND       P01415	// W450 메인파트
OR LOAD
AND LOAD
MOV       2 D001311	// W450 파트램프 상태
// //////파트이미지 화면전환
; L114
LOADP     M01314	// W450 파트이상
ORP       M01315	// W450 차종이상
ORP       M0131D	// W450 파트센서 체크 이상
ORP       M0131E	// W450 슬라이드 안착이상
MOVP      117 D015010	// OP2 Touch Display Change
; L118
LOADP     M0131C	// W450 유니트 센서이상
MOVP      17 D015010	// OP2 Touch Display Change
; L119
END

PROGRAM MAIN_STN15_W(M1500) (task: 스캔 프로그램)

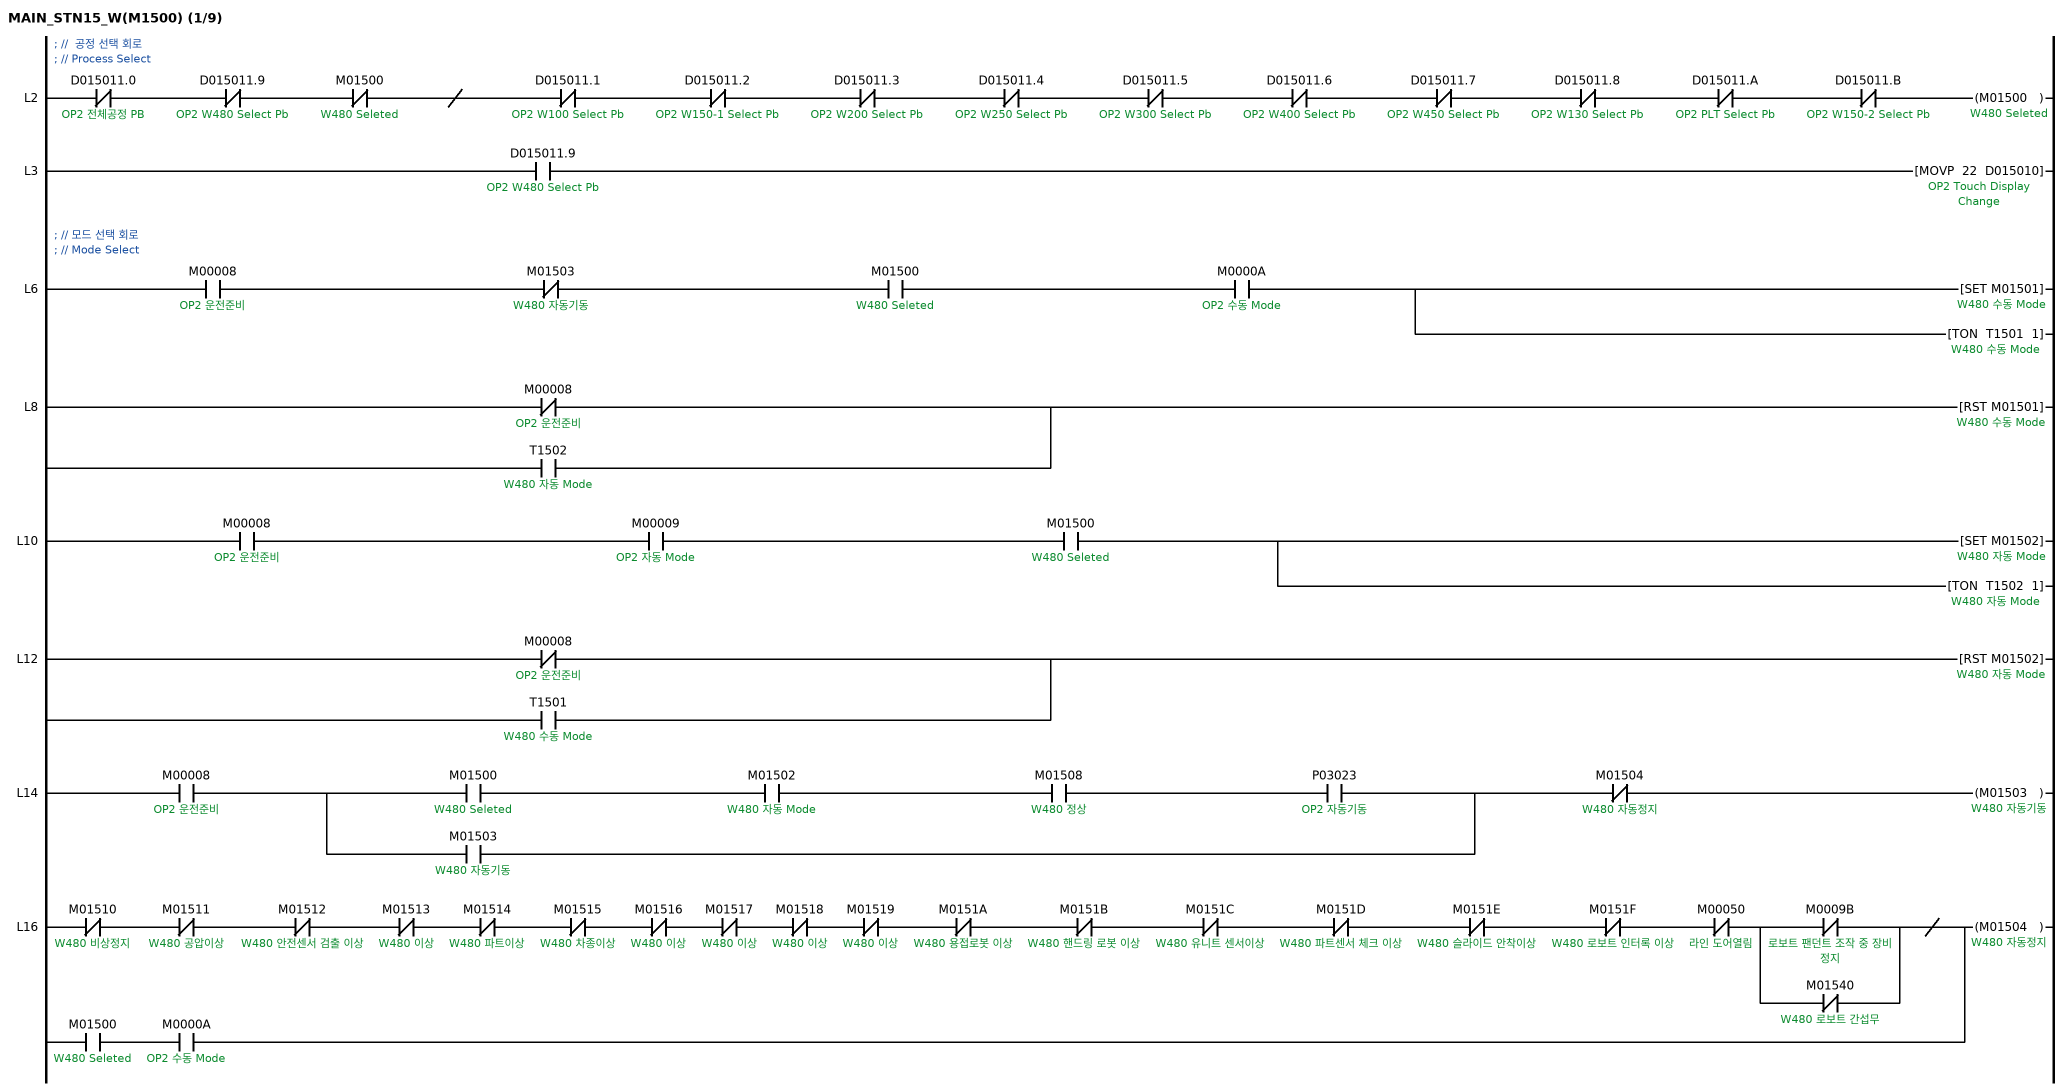
//   //  공정 선택 회로
//   // Process Select
; L2
LOAD NOT  D015011.0	// OP2 전체공정 PB
AND NOT   D015011.9	// OP2 W480 Select Pb
AND NOT   M01500	// W480 Seleted
NOT
AND NOT   D015011.1	// OP2 W100 Select Pb
AND NOT   D015011.2	// OP2 W150-1 Select Pb
AND NOT   D015011.3	// OP2 W200 Select Pb
AND NOT   D015011.4	// OP2 W250 Select Pb
AND NOT   D015011.5	// OP2 W300 Select Pb
AND NOT   D015011.6	// OP2 W400 Select Pb
AND NOT   D015011.7	// OP2 W450 Select Pb
AND NOT   D015011.8	// OP2 W130 Select Pb
AND NOT   D015011.A	// OP2 PLT Select Pb
AND NOT   D015011.B	// OP2 W150-2 Select Pb
OUT       M01500	// W480 Seleted
; L3
LOAD      D015011.9	// OP2 W480 Select Pb
MOVP      22 D015010	// OP2 Touch Display Change
// // 모드 선택 회로
//   // Mode Select
; L6
LOAD      M00008	// OP2 운전준비
AND NOT   M01503	// W480 자동기동
AND       M01500	// W480 Seleted
AND       M0000A	// OP2 수동 Mode
SET       M01501	// W480 수동 Mode
TON       T1501 1	// W480 수동 Mode
; L8
LOAD NOT  M00008	// OP2 운전준비
OR        T1502	// W480 자동 Mode
RST       M01501	// W480 수동 Mode
; L10
LOAD      M00008	// OP2 운전준비
AND       M00009	// OP2 자동 Mode
AND       M01500	// W480 Seleted
SET       M01502	// W480 자동 Mode
TON       T1502 1	// W480 자동 Mode
; L12
LOAD NOT  M00008	// OP2 운전준비
OR        T1501	// W480 수동 Mode
RST       M01502	// W480 자동 Mode
; L14
LOAD      M00008	// OP2 운전준비
LOAD      M01500	// W480 Seleted
AND       M01502	// W480 자동 Mode
AND       M01508	// W480 정상
AND       P03023	// OP2 자동기동
OR        M01503	// W480 자동기동
AND LOAD
AND NOT   M01504	// W480 자동정지
OUT       M01503	// W480 자동기동
; L16
LOAD NOT  M01510	// W480 비상정지
AND NOT   M01511	// W480 공압이상
AND NOT   M01512	// W480 안전센서 검출 이상
AND NOT   M01513	// W480 이상
AND NOT   M01514	// W480 파트이상
AND NOT   M01515	// W480 차종이상
AND NOT   M01516	// W480 이상
AND NOT   M01517	// W480 이상
AND NOT   M01518	// W480 이상
AND NOT   M01519	// W480 이상
AND NOT   M0151A	// W480 용접로봇 이상
AND NOT   M0151B	// W480 핸드링 로봇 이상
AND NOT   M0151C	// W480 유니트 센서이상
AND NOT   M0151D	// W480 파트센서 체크 이상
AND NOT   M0151E	// W480 슬라이드 안착이상
AND NOT   M0151F	// W480 로보트 인터록 이상
AND NOT   M00050	// 라인 도어열림
LOAD NOT  M0009B	// 로보트 팬던트 조작 중 장비 정지
OR NOT    M01540	// W480 로보트 간섭무
AND LOAD
NOT
LOAD      M01500	// W480 Seleted
AND       M0000A	// OP2 수동 Mode
OR LOAD
OUT       M01504	// W480 자동정지

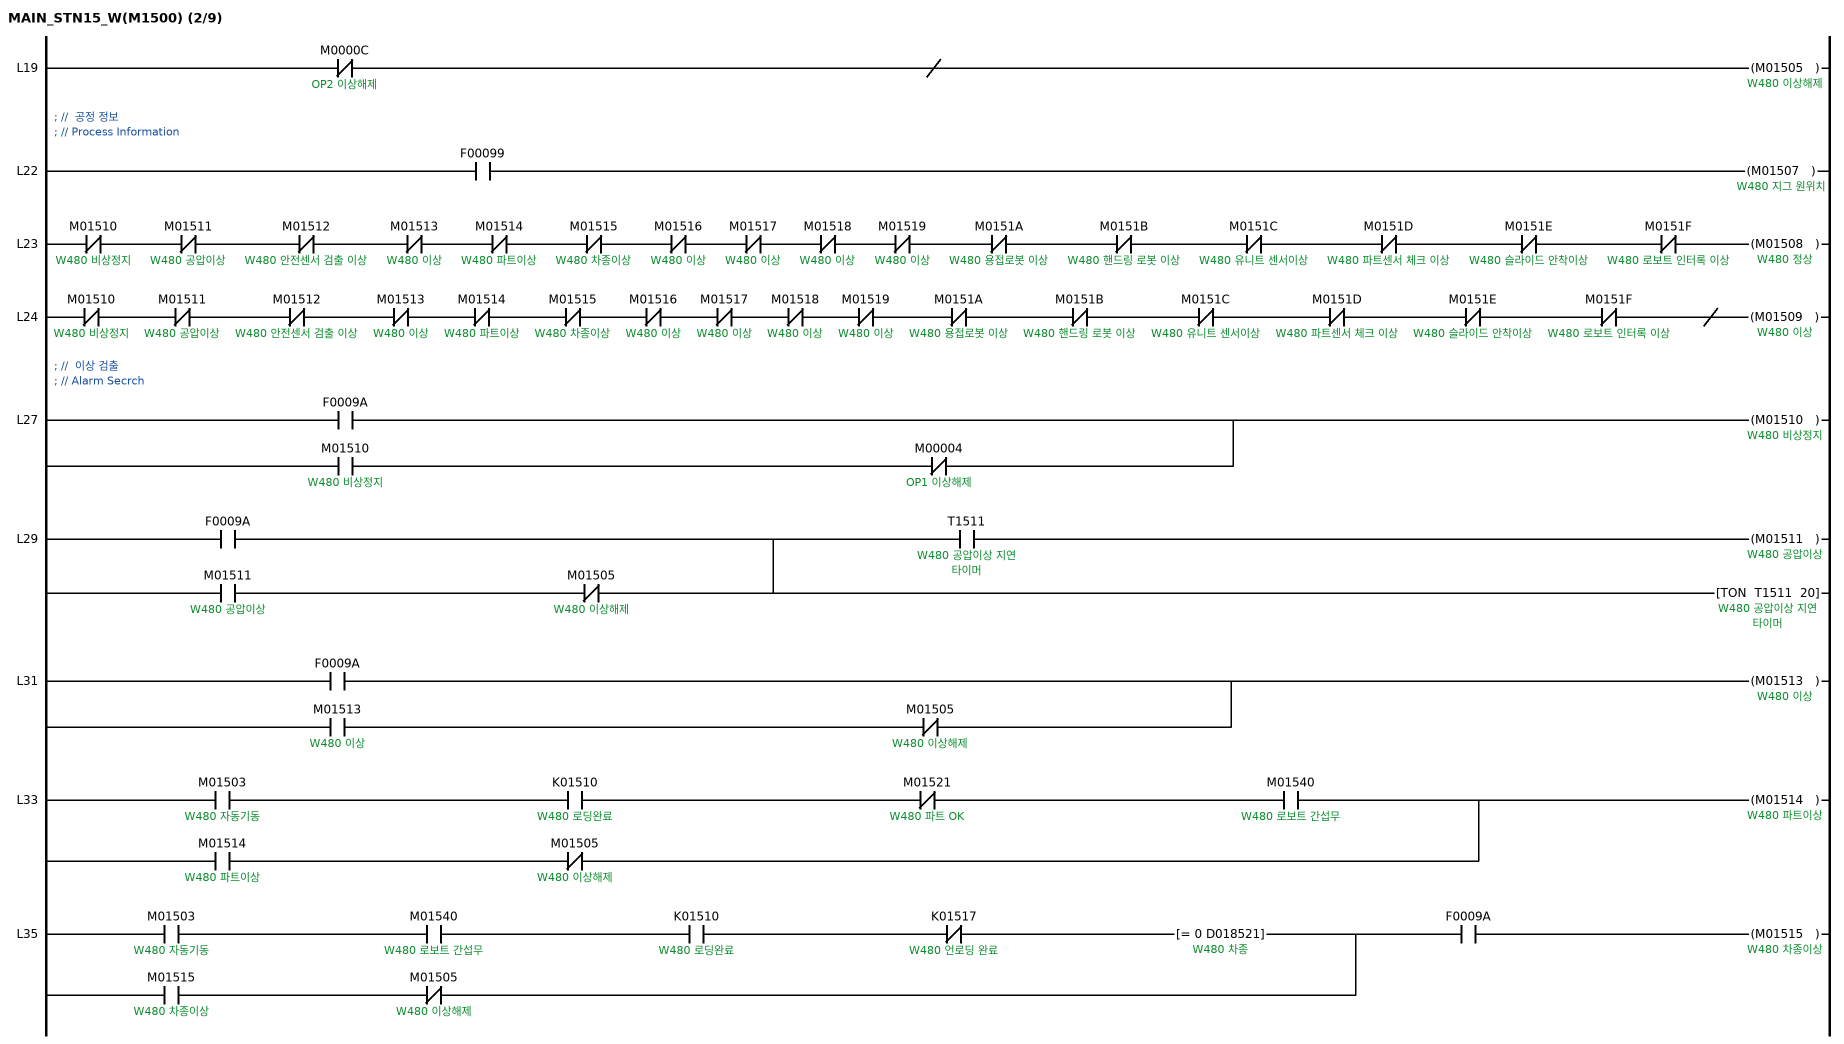
; L19
LOAD NOT  M0000C	// OP2 이상해제
NOT
OUT       M01505	// W480 이상해제
//   //  공정 정보
//   // Process Information
; L22
LOAD      F00099
OUT       M01507	// W480 지그 원위치
; L23
LOAD NOT  M01510	// W480 비상정지
AND NOT   M01511	// W480 공압이상
AND NOT   M01512	// W480 안전센서 검출 이상
AND NOT   M01513	// W480 이상
AND NOT   M01514	// W480 파트이상
AND NOT   M01515	// W480 차종이상
AND NOT   M01516	// W480 이상
AND NOT   M01517	// W480 이상
AND NOT   M01518	// W480 이상
AND NOT   M01519	// W480 이상
AND NOT   M0151A	// W480 용접로봇 이상
AND NOT   M0151B	// W480 핸드링 로봇 이상
AND NOT   M0151C	// W480 유니트 센서이상
AND NOT   M0151D	// W480 파트센서 체크 이상
AND NOT   M0151E	// W480 슬라이드 안착이상
AND NOT   M0151F	// W480 로보트 인터록 이상
OUT       M01508	// W480 정상
; L24
LOAD NOT  M01510	// W480 비상정지
AND NOT   M01511	// W480 공압이상
AND NOT   M01512	// W480 안전센서 검출 이상
AND NOT   M01513	// W480 이상
AND NOT   M01514	// W480 파트이상
AND NOT   M01515	// W480 차종이상
AND NOT   M01516	// W480 이상
AND NOT   M01517	// W480 이상
AND NOT   M01518	// W480 이상
AND NOT   M01519	// W480 이상
AND NOT   M0151A	// W480 용접로봇 이상
AND NOT   M0151B	// W480 핸드링 로봇 이상
AND NOT   M0151C	// W480 유니트 센서이상
AND NOT   M0151D	// W480 파트센서 체크 이상
AND NOT   M0151E	// W480 슬라이드 안착이상
AND NOT   M0151F	// W480 로보트 인터록 이상
NOT
OUT       M01509	// W480 이상
//   //  이상 검출
//   // Alarm Secrch
; L27
LOAD      F0009A
LOAD      M01510	// W480 비상정지
AND NOT   M00004	// OP1 이상해제
OR LOAD
OUT       M01510	// W480 비상정지
; L29
LOAD      F0009A
LOAD      M01511	// W480 공압이상
AND NOT   M01505	// W480 이상해제
OR LOAD
MPUSH
AND       T1511	// W480 공압이상 지연 타이머
OUT       M01511	// W480 공압이상
MPOP
TON       T1511 20	// W480 공압이상 지연 타이머
; L31
LOAD      F0009A
LOAD      M01513	// W480 이상
AND NOT   M01505	// W480 이상해제
OR LOAD
OUT       M01513	// W480 이상
; L33
LOAD      M01503	// W480 자동기동
AND       K01510	// W480 로딩완료
AND NOT   M01521	// W480 파트 OK
AND       M01540	// W480 로보트 간섭무
LOAD      M01514	// W480 파트이상
AND NOT   M01505	// W480 이상해제
OR LOAD
OUT       M01514	// W480 파트이상
; L35
LOAD      M01503	// W480 자동기동
AND       M01540	// W480 로보트 간섭무
AND       K01510	// W480 로딩완료
AND NOT   K01517	// W480 언로딩 완료
AND=      0 D018521	// W480 차종
LOAD      M01515	// W480 차종이상
AND NOT   M01505	// W480 이상해제
OR LOAD
AND       F0009A
OUT       M01515	// W480 차종이상

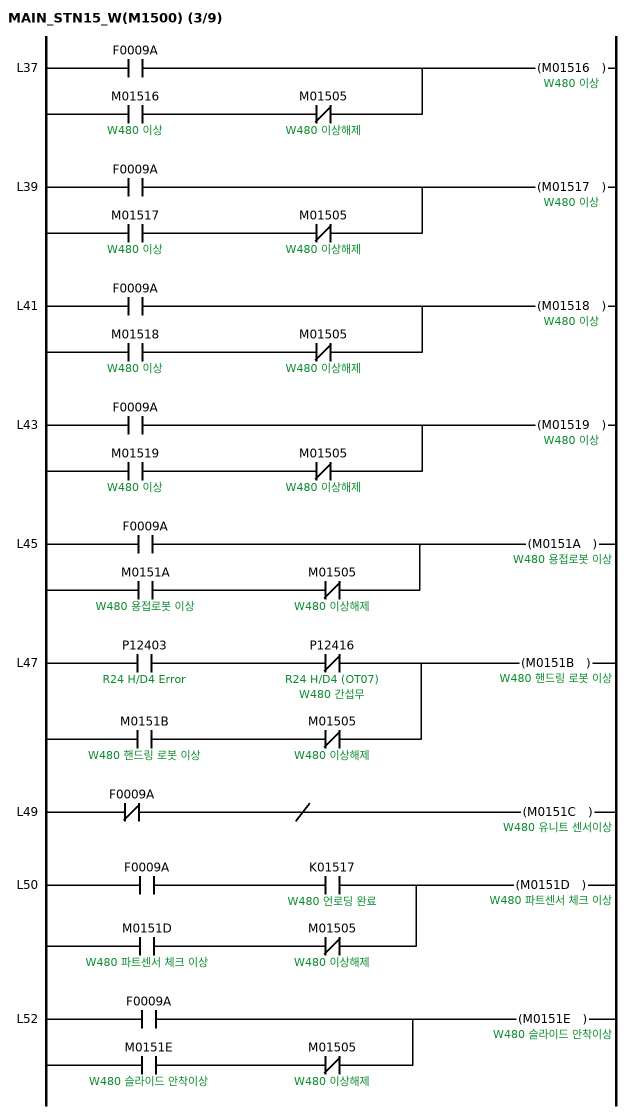
; L37
LOAD      F0009A
LOAD      M01516	// W480 이상
AND NOT   M01505	// W480 이상해제
OR LOAD
OUT       M01516	// W480 이상
; L39
LOAD      F0009A
LOAD      M01517	// W480 이상
AND NOT   M01505	// W480 이상해제
OR LOAD
OUT       M01517	// W480 이상
; L41
LOAD      F0009A
LOAD      M01518	// W480 이상
AND NOT   M01505	// W480 이상해제
OR LOAD
OUT       M01518	// W480 이상
; L43
LOAD      F0009A
LOAD      M01519	// W480 이상
AND NOT   M01505	// W480 이상해제
OR LOAD
OUT       M01519	// W480 이상
; L45
LOAD      F0009A
LOAD      M0151A	// W480 용접로봇 이상
AND NOT   M01505	// W480 이상해제
OR LOAD
OUT       M0151A	// W480 용접로봇 이상
; L47
LOAD      P12403	// R24 H/D4 Error
AND NOT   P12416	// R24 H/D4 (OT07) W480 간섭무
LOAD      M0151B	// W480 핸드링 로봇 이상
AND NOT   M01505	// W480 이상해제
OR LOAD
OUT       M0151B	// W480 핸드링 로봇 이상
; L49
LOAD NOT  F0009A
NOT
OUT       M0151C	// W480 유니트 센서이상
; L50
LOAD      F0009A
AND       K01517	// W480 언로딩 완료
LOAD      M0151D	// W480 파트센서 체크 이상
AND NOT   M01505	// W480 이상해제
OR LOAD
OUT       M0151D	// W480 파트센서 체크 이상
; L52
LOAD      F0009A
LOAD      M0151E	// W480 슬라이드 안착이상
AND NOT   M01505	// W480 이상해제
OR LOAD
OUT       M0151E	// W480 슬라이드 안착이상

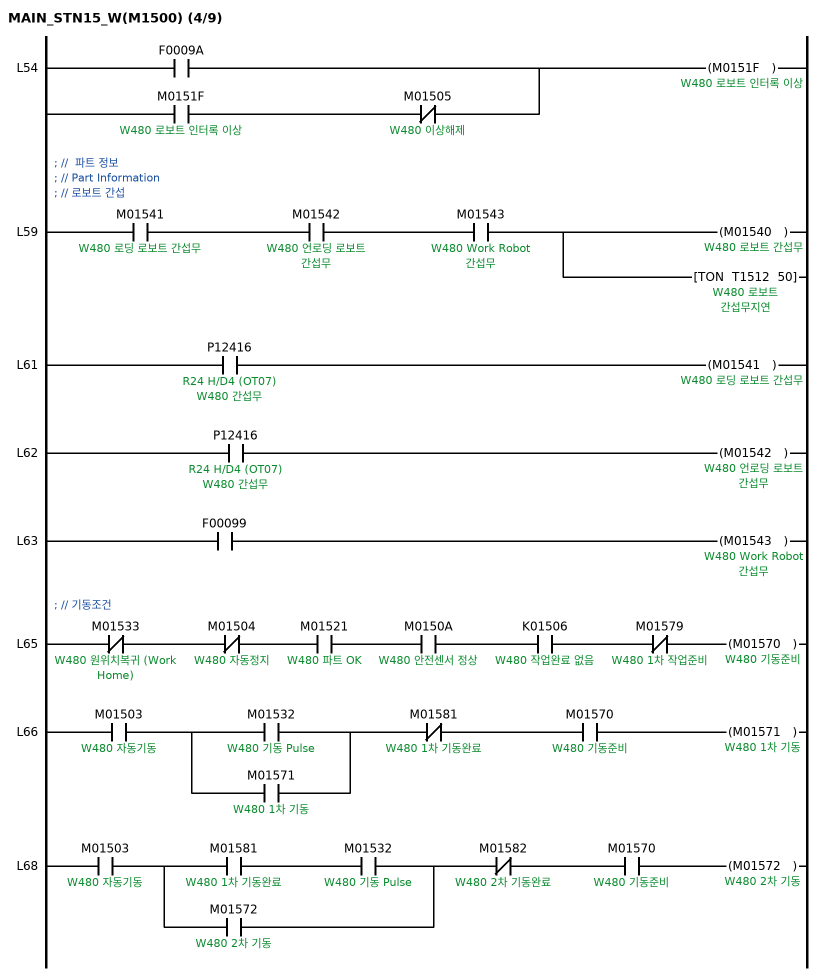
; L54
LOAD      F0009A
LOAD      M0151F	// W480 로보트 인터록 이상
AND NOT   M01505	// W480 이상해제
OR LOAD
OUT       M0151F	// W480 로보트 인터록 이상
//   //  파트 정보
//   // Part Information
//   // 로보트 간섭
; L59
LOAD      M01541	// W480 로딩 로보트 간섭무
AND       M01542	// W480 언로딩 로보트 간섭무
AND       M01543	// W480 Work Robot 간섭무
OUT       M01540	// W480 로보트 간섭무
TON       T1512 50	// W480 로보트 간섭무지연
; L61
LOAD      P12416	// R24 H/D4 (OT07) W480 간섭무
OUT       M01541	// W480 로딩 로보트 간섭무
; L62
LOAD      P12416	// R24 H/D4 (OT07) W480 간섭무
OUT       M01542	// W480 언로딩 로보트 간섭무
; L63
LOAD      F00099
OUT       M01543	// W480 Work Robot 간섭무
//   // 기동조건
; L65
LOAD NOT  M01533	// W480 원위치복귀 (Work Home)
AND NOT   M01504	// W480 자동정지
AND       M01521	// W480 파트 OK
AND       M0150A	// W480 안전센서 정상
AND       K01506	// W480 작업완료 없음
AND NOT   M01579	// W480 1차 작업준비
OUT       M01570	// W480 기동준비
; L66
LOAD      M01503	// W480 자동기동
LOAD      M01532	// W480 기동 Pulse
OR        M01571	// W480 1차 기동
AND LOAD
AND NOT   M01581	// W480 1차 기동완료
AND       M01570	// W480 기동준비
OUT       M01571	// W480 1차 기동
; L68
LOAD      M01503	// W480 자동기동
LOAD      M01581	// W480 1차 기동완료
AND       M01532	// W480 기동 Pulse
OR        M01572	// W480 2차 기동
AND LOAD
AND NOT   M01582	// W480 2차 기동완료
AND       M01570	// W480 기동준비
OUT       M01572	// W480 2차 기동

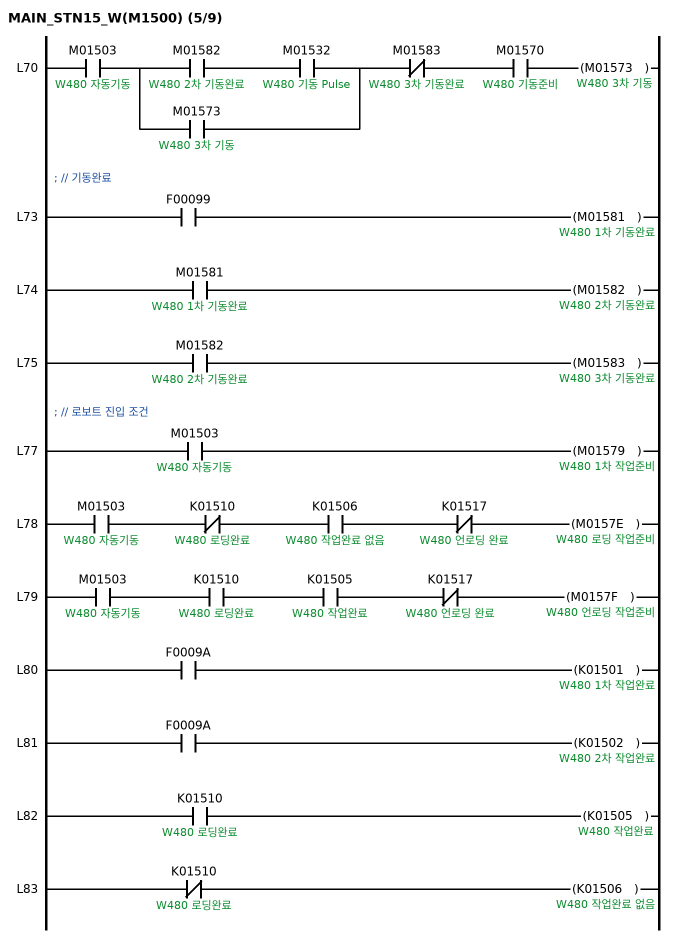
; L70
LOAD      M01503	// W480 자동기동
LOAD      M01582	// W480 2차 기동완료
AND       M01532	// W480 기동 Pulse
OR        M01573	// W480 3차 기동
AND LOAD
AND NOT   M01583	// W480 3차 기동완료
AND       M01570	// W480 기동준비
OUT       M01573	// W480 3차 기동
//   // 기동완료
; L73
LOAD      F00099
OUT       M01581	// W480 1차 기동완료
; L74
LOAD      M01581	// W480 1차 기동완료
OUT       M01582	// W480 2차 기동완료
; L75
LOAD      M01582	// W480 2차 기동완료
OUT       M01583	// W480 3차 기동완료
//   // 로보트 진입 조건
; L77
LOAD      M01503	// W480 자동기동
OUT       M01579	// W480 1차 작업준비
; L78
LOAD      M01503	// W480 자동기동
AND NOT   K01510	// W480 로딩완료
AND       K01506	// W480 작업완료 없음
AND NOT   K01517	// W480 언로딩 완료
OUT       M0157E	// W480 로딩 작업준비
; L79
LOAD      M01503	// W480 자동기동
AND       K01510	// W480 로딩완료
AND       K01505	// W480 작업완료
AND NOT   K01517	// W480 언로딩 완료
OUT       M0157F	// W480 언로딩 작업준비
; L80
LOAD      F0009A
OUT       K01501	// W480 1차 작업완료
; L81
LOAD      F0009A
OUT       K01502	// W480 2차 작업완료
; L82
LOAD      K01510	// W480 로딩완료
OUT       K01505	// W480 작업완료
; L83
LOAD NOT  K01510	// W480 로딩완료
OUT       K01506	// W480 작업완료 없음

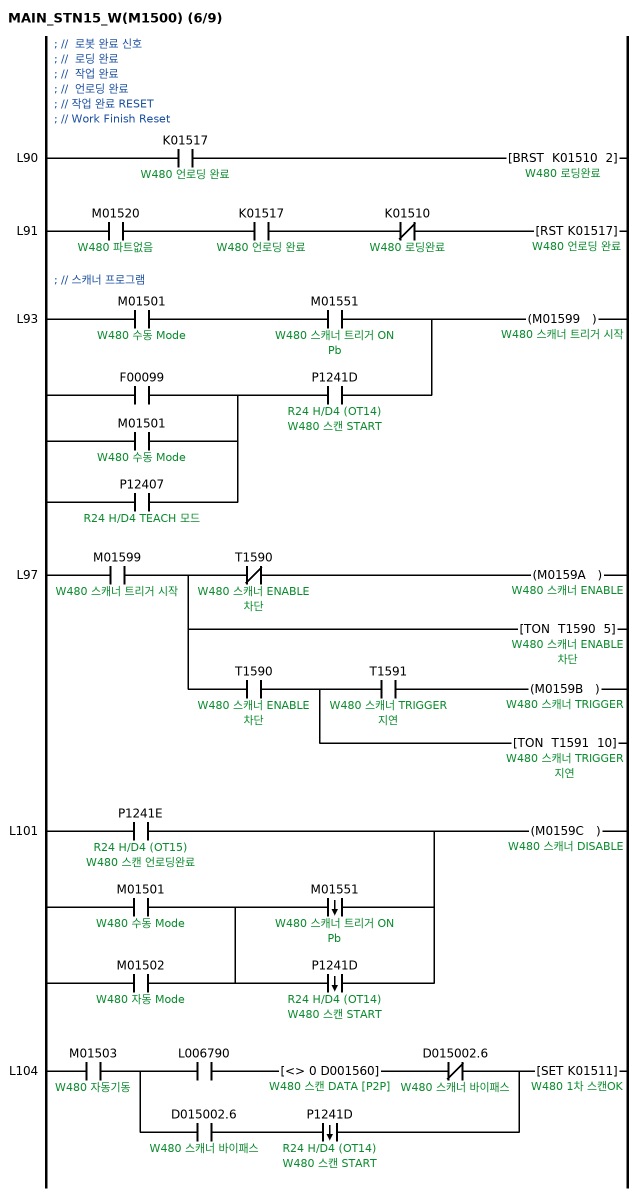
//   //  로봇 완료 신호
//   //  로딩 완료
//   //  작업 완료
//   //  언로딩 완료
//     // 작업 완료 RESET
//   // Work Finish Reset
; L90
LOAD      K01517	// W480 언로딩 완료
BRST      K01510 2	// W480 로딩완료
; L91
LOAD      M01520	// W480 파트없음
AND       K01517	// W480 언로딩 완료
AND NOT   K01510	// W480 로딩완료
RST       K01517	// W480 언로딩 완료
//   // 스캐너 프로그램
; L93
LOAD      M01501	// W480 수동 Mode
AND       M01551	// W480 스캐너 트리거 ON Pb
LOAD      F00099
OR        M01501	// W480 수동 Mode
OR        P12407	// R24 H/D4 TEACH 모드
AND       P1241D	// R24 H/D4 (OT14) W480 스캔 START
OR LOAD
OUT       M01599	// W480 스캐너 트리거 시작
; L97
LOAD      M01599	// W480 스캐너 트리거 시작
MPUSH
AND NOT   T1590	// W480 스캐너 ENABLE 차단
OUT       M0159A	// W480 스캐너 ENABLE
MPOP
TON       T1590 5	// W480 스캐너 ENABLE 차단
AND       T1590	// W480 스캐너 ENABLE 차단
MPUSH
AND       T1591	// W480 스캐너 TRIGGER 지연
OUT       M0159B	// W480 스캐너 TRIGGER
MPOP
TON       T1591 10	// W480 스캐너 TRIGGER 지연
; L101
LOAD      P1241E	// R24 H/D4 (OT15) W480 스캔 언로딩완료
LOAD      M01501	// W480 수동 Mode
OR        M01502	// W480 자동 Mode
LOADN     M01551	// W480 스캐너 트리거 ON Pb
ORN       P1241D	// R24 H/D4 (OT14) W480 스캔 START
AND LOAD
OR LOAD
OUT       M0159C	// W480 스캐너 DISABLE
; L104
LOAD      M01503	// W480 자동기동
LOAD      L006790
AND<>     0 D001560	// W480 스캔 DATA [P2P]
AND NOT   D015002.6	// W480 스캐너 바이패스
LOAD      D015002.6	// W480 스캐너 바이패스
ANDN      P1241D	// R24 H/D4 (OT14) W480 스캔 START
OR LOAD
AND LOAD
SET       K01511	// W480 1차 스캔OK

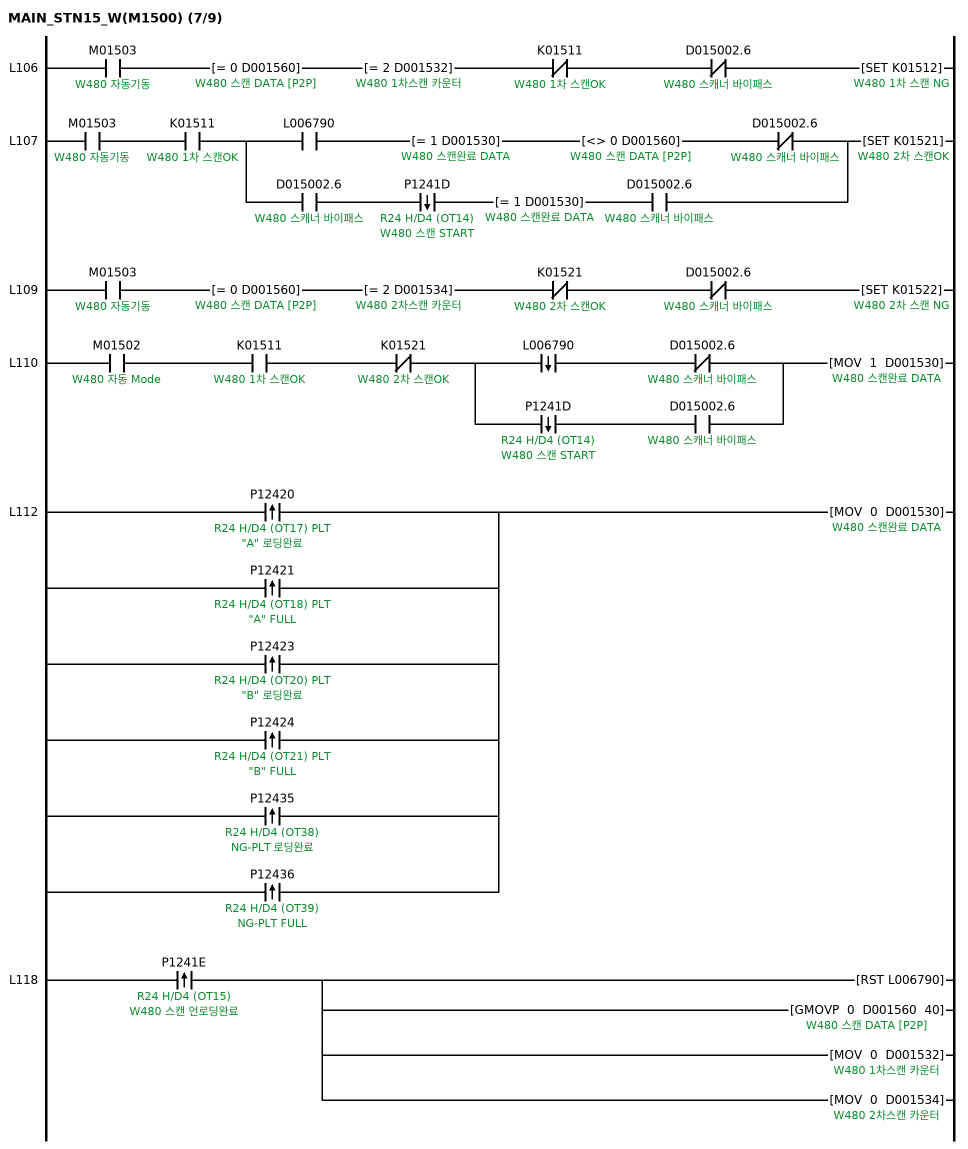
; L106
LOAD      M01503	// W480 자동기동
AND=      0 D001560	// W480 스캔 DATA [P2P]
AND=      2 D001532	// W480 1차스캔 카운터
AND NOT   K01511	// W480 1차 스캔OK
AND NOT   D015002.6	// W480 스캐너 바이패스
SET       K01512	// W480 1차 스캔 NG
; L107
LOAD      M01503	// W480 자동기동
AND       K01511	// W480 1차 스캔OK
LOAD      L006790
AND=      1 D001530	// W480 스캔완료 DATA
AND<>     0 D001560	// W480 스캔 DATA [P2P]
AND NOT   D015002.6	// W480 스캐너 바이패스
LOAD      D015002.6	// W480 스캐너 바이패스
ANDN      P1241D	// R24 H/D4 (OT14) W480 스캔 START
AND=      1 D001530	// W480 스캔완료 DATA
AND       D015002.6	// W480 스캐너 바이패스
OR LOAD
AND LOAD
SET       K01521	// W480 2차 스캔OK
; L109
LOAD      M01503	// W480 자동기동
AND=      0 D001560	// W480 스캔 DATA [P2P]
AND=      2 D001534	// W480 2차스캔 카운터
AND NOT   K01521	// W480 2차 스캔OK
AND NOT   D015002.6	// W480 스캐너 바이패스
SET       K01522	// W480 2차 스캔 NG
; L110
LOAD      M01502	// W480 자동 Mode
AND       K01511	// W480 1차 스캔OK
AND NOT   K01521	// W480 2차 스캔OK
LOADN     L006790
AND NOT   D015002.6	// W480 스캐너 바이패스
LOADN     P1241D	// R24 H/D4 (OT14) W480 스캔 START
AND       D015002.6	// W480 스캐너 바이패스
OR LOAD
AND LOAD
MOV       1 D001530	// W480 스캔완료 DATA
; L112
LOADP     P12420	// R24 H/D4 (OT17) PLT "A" 로딩완료
ORP       P12421	// R24 H/D4 (OT18) PLT "A" FULL
ORP       P12423	// R24 H/D4 (OT20) PLT "B" 로딩완료
ORP       P12424	// R24 H/D4 (OT21) PLT "B" FULL
ORP       P12435	// R24 H/D4 (OT38) NG-PLT 로딩완료
ORP       P12436	// R24 H/D4 (OT39) NG-PLT FULL
MOV       0 D001530	// W480 스캔완료 DATA
; L118
LOADP     P1241E	// R24 H/D4 (OT15) W480 스캔 언로딩완료
RST       L006790
GMOVP     0 D001560 40	// W480 스캔 DATA [P2P]
MOV       0 D001532	// W480 1차스캔 카운터
MOV       0 D001534	// W480 2차스캔 카운터

